LIN {X 0,Y 520.453,Z 702.53,A -85,B 0,C 180,E1 4696.9,E2 4696.9} C_VEL
LIN {X 0,Y 520.349,Z 702.53,A -85,B 0,C 180,E1 4702.128,E2 4702.128} C_VEL
LIN {X 0,Y 520.208,Z 702.53,A -85,B 0,C 180,E1 4707.632,E2 4707.632} C_VEL
LIN {X 0,Y 520.173,Z 702.53,A -85,B 0,C 180,E1 4713.424,E2 4713.424} C_VEL
LIN {X 0,Y 520.246,Z 702.53,A -85,B 0,C 180,E1 4719.624,E2 4719.624} C_VEL
LIN {X 0,Y 520.141,Z 702.53,A -85,B 0,C 180,E1 4725.871,E2 4725.871} C_VEL
LIN {X 0,Y 520.098,Z 702.53,A -85,B 0,C 180,E1 4731.533,E2 4731.533} C_VEL
LIN {X 0,Y 520.321,Z 702.53,A -85,B 0,C 180,E1 4737.206,E2 4737.206} C_VEL
LIN {X 0,Y 520.267,Z 702.53,A -85,B 0,C 180,E1 4742.35,E2 4742.35} C_VEL
LIN {X 0,Y 520.358,Z 702.53,A -85,B 0,C 180,E1 4748.054,E2 4748.054} C_VEL
LIN {X 0,Y 520.437,Z 702.53,A -85,B 0,C 180,E1 4753.145,E2 4753.145} C_VEL
LIN {X 0,Y 520.522,Z 702.53,A -85,B 0,C 180,E1 4758.292,E2 4758.292} C_VEL
LIN {X 0,Y 520.587,Z 702.53,A -85,B 0,C 180,E1 4763.342,E2 4763.342} C_VEL
LIN {X 0,Y 520.67,Z 703.242,A -85,B 0,C 180,E1 4767.374,E2 4767.374} C_VEL
LIN {X 0,Y 530.204,Z 730.276,A -85,B 0,C 180,E1 4768.601,E2 4768.601} C_VEL
LIN {X 0,Y 528.889,Z 767.403,A -85,B 0,C 180,E1 4769.944,E2 4769.944} C_VEL
LIN {X 0,Y 527.056,Z 803.071,A -85,B 0,C 180,E1 4771.949,E2 4771.949} C_VEL
LIN {X 0,Y 525.109,Z 835.334,A -85,B 0,C 180,E1 4774.533,E2 4774.533} C_VEL
LIN {X 0,Y 523.491,Z 864.071,A -85,B 0,C 180,E1 4777.662,E2 4777.662} C_VEL
LIN {X 0,Y 522.246,Z 888.252,A -85,B 0,C 180,E1 4781.228,E2 4781.228} C_VEL
LIN {X 0,Y 521.421,Z 907.192,A -85,B 0,C 180,E1 4785.098,E2 4785.098} C_VEL
LIN {X 0,Y 521.133,Z 919.028,A -85,B 0,C 180,E1 4788.574,E2 4788.574} C_VEL
LIN {X 0,Y 520.904,Z 926.713,A -85,B 0,C 180,E1 4792.124,E2 4792.124} C_VEL
LIN {X 0,Y 520.609,Z 930.33,A -85,B 0,C 180,E1 4796.089,E2 4796.089} C_VEL
LIN {X 0,Y 520.787,Z 928.438,A -85,B 0,C 180,E1 4800.509,E2 4800.509} C_VEL
LIN {X 0,Y 521.135,Z 920.633,A -85,B 0,C 180,E1 4804.748,E2 4804.748} C_VEL
LIN {X 0,Y 521.384,Z 907.878,A -85,B 0,C 180,E1 4808.645,E2 4808.645} C_VEL
LIN {X 0,Y 522.078,Z 890.326,A -85,B 0,C 180,E1 4812.316,E2 4812.316} C_VEL
LIN {X 0,Y 523.248,Z 867.61,A -85,B 0,C 180,E1 4815.79,E2 4815.79} C_VEL
LIN {X 0,Y 524.928,Z 839.521,A -85,B 0,C 180,E1 4818.979,E2 4818.979} C_VEL
LIN {X 0,Y 526.831,Z 807.399,A -85,B 0,C 180,E1 4821.654,E2 4821.654} C_VEL
LIN {X 0,Y 528.689,Z 772.934,A -85,B 0,C 180,E1 4823.704,E2 4823.704} C_VEL
LIN {X 0,Y 530.241,Z 736.63,A -85,B 0,C 180,E1 4825.119,E2 4825.119} C_VEL
LIN {X 0,Y 529.84,Z 727.033,A -85,B 0,C 180,E1 4825.43,E2 4825.43} C_VEL
LIN {X 0,Y 520.271,Z 702.53,A -85,B 0,C 180,E1 4826.686,E2 4826.686} C_VEL
LIN {X 0,Y 520.292,Z 702.53,A -85,B 0,C 180,E1 4832.373,E2 4832.373} C_VEL
LIN {X 0,Y 520.403,Z 702.53,A -85,B 0,C 180,E1 4838.112,E2 4838.112} C_VEL
LIN {X 0,Y 520.549,Z 702.53,A -85,B 0,C 180,E1 4843.167,E2 4843.167} C_VEL
LIN {X 0,Y 520.567,Z 702.53,A -85,B 0,C 180,E1 4848.309,E2 4848.309} C_VEL
LIN {X 0,Y 520.603,Z 702.53,A -85,B 0,C 180,E1 4853.357,E2 4853.357} C_VEL
LIN {X 0,Y 520.62,Z 702.53,A -85,B 0,C 180,E1 4858.353,E2 4858.353} C_VEL
LIN {X 0,Y 520.671,Z 702.53,A -85,B 0,C 180,E1 4863.336,E2 4863.336} C_VEL
LIN {X 0,Y 520.512,Z 702.53,A -85,B 0,C 180,E1 4868.346,E2 4868.346} C_VEL
LIN {X 0,Y 520.449,Z 702.53,A -85,B 0,C 180,E1 4873.423,E2 4873.423} C_VEL
LIN {X 0,Y 520.367,Z 702.53,A -85,B 0,C 180,E1 4878.611,E2 4878.611} C_VEL
LIN {X 0,Y 520.283,Z 702.53,A -85,B 0,C 180,E1 4883.966,E2 4883.966} C_VEL
LIN {X 0,Y 520.16,Z 702.53,A -85,B 0,C 180,E1 4889.558,E2 4889.558} C_VEL
LIN {X 0,Y 520.063,Z 702.53,A -85,B 0,C 180,E1 4894.193,E2 4894.193} C_VEL
LIN {X 0,Y 516.119,Z 702.53,A -85,B 0,C 180,E1 4896.079,E2 4896.079} C_VEL
LIN {X 0,Y 512.277,Z 702.53,A -85,B 0,C 180,E1 4897.994,E2 4897.994} C_VEL
LIN {X 0,Y 512.218,Z 702.53,A -85,B 0,C 180,E1 4902.662,E2 4902.662} C_VEL
LIN {X 0,Y 512.145,Z 702.53,A -85,B 0,C 180,E1 4907.449,E2 4907.449} C_VEL
LIN {X 0,Y 512.253,Z 702.53,A -85,B 0,C 180,E1 4914.109,E2 4914.109} C_VEL
LIN {X 0,Y 527.514,Z 735.275,A -85,B 0,C 180,E1 4915.852,E2 4915.852} C_VEL
LIN {X 0,Y 526.665,Z 780.172,A -85,B 0,C 180,E1 4916.724,E2 4916.724} C_VEL
LIN {X 0,Y 525.012,Z 817.63,A -85,B 0,C 180,E1 4918.058,E2 4918.058} C_VEL
LIN {X 0,Y 522.673,Z 854.221,A -85,B 0,C 180,E1 4920.016,E2 4920.016} C_VEL
LIN {X 0,Y 520.021,Z 889.901,A -85,B 0,C 180,E1 4922.686,E2 4922.686} C_VEL
LIN {X 0,Y 517.692,Z 920.346,A -85,B 0,C 180,E1 4925.724,E2 4925.724} C_VEL
LIN {X 0,Y 515.734,Z 947.246,A -85,B 0,C 180,E1 4929.22,E2 4929.22} C_VEL
LIN {X 0,Y 514.274,Z 970.267,A -85,B 0,C 180,E1 4933.156,E2 4933.156} C_VEL
LIN {X 0,Y 513.457,Z 987.982,A -85,B 0,C 180,E1 4937.266,E2 4937.266} C_VEL
LIN {X 0,Y 513.159,Z 1000.677,A -85,B 0,C 180,E1 4941.545,E2 4941.545} C_VEL
LIN {X 0,Y 512.986,Z 1006.957,A -85,B 0,C 180,E1 4944.937,E2 4944.937} C_VEL
LIN {X 0,Y 513.01,Z 1010.088,A -85,B 0,C 180,E1 4948.314,E2 4948.314} C_VEL
LIN {X 0,Y 513.121,Z 1010.089,A -85,B 0,C 180,E1 4951.685,E2 4951.685} C_VEL
LIN {X 0,Y 513.106,Z 1005.755,A -85,B 0,C 180,E1 4955.908,E2 4955.908} C_VEL
LIN {X 0,Y 513.225,Z 996.305,A -85,B 0,C 180,E1 4960.161,E2 4960.161} C_VEL
LIN {X 0,Y 513.729,Z 982.23,A -85,B 0,C 180,E1 4964.223,E2 4964.223} C_VEL
LIN {X 0,Y 514.773,Z 962.39,A -85,B 0,C 180,E1 4968.322,E2 4968.322} C_VEL
LIN {X 0,Y 516.496,Z 936.317,A -85,B 0,C 180,E1 4972.322,E2 4972.322} C_VEL
LIN {X 0,Y 518.843,Z 905.455,A -85,B 0,C 180,E1 4975.866,E2 4975.866} C_VEL
LIN {X 0,Y 521.362,Z 871.934,A -85,B 0,C 180,E1 4978.763,E2 4978.763} C_VEL
LIN {X 0,Y 523.868,Z 836.553,A -85,B 0,C 180,E1 4981.015,E2 4981.015} C_VEL
LIN {X 0,Y 525.939,Z 799.077,A -85,B 0,C 180,E1 4982.679,E2 4982.679} C_VEL
LIN {X 0,Y 527.422,Z 761.468,A -85,B 0,C 180,E1 4983.701,E2 4983.701} C_VEL
LIN {X 0,Y 526.932,Z 733.943,A -85,B 0,C 180,E1 4984.213,E2 4984.213} C_VEL
LIN {X 0,Y 512.224,Z 702.53,A -85,B 0,C 180,E1 4985.89,E2 4985.89} C_VEL
LIN {X 0,Y 512.283,Z 702.53,A -85,B 0,C 180,E1 4990.395,E2 4990.395} C_VEL
LIN {X 0,Y 512.226,Z 702.53,A -85,B 0,C 180,E1 4995,E2 4995} C_VEL
LIN {X 0,Y 512.163,Z 702.53,A -85,B 0,C 180,E1 5000.001,E2 5000.001} C_VEL
LIN {X 0,Y 512.28,Z 702.53,A -85,B 0,C 180,E1 5005.959,E2 5005.959} C_VEL
LIN {X 0,Y 512.335,Z 702.53,A -85,B 0,C 180,E1 5011.876,E2 5011.876} C_VEL
LIN {X 0,Y 512.348,Z 702.53,A -85,B 0,C 180,E1 5017.478,E2 5017.478} C_VEL
LIN {X 0,Y 512.571,Z 702.53,A -85,B 0,C 180,E1 5022.868,E2 5022.868} C_VEL
LIN {X 0,Y 512.624,Z 702.53,A -85,B 0,C 180,E1 5028.097,E2 5028.097} C_VEL
LIN {X 0,Y 512.715,Z 702.53,A -85,B 0,C 180,E1 5033.227,E2 5033.227} C_VEL
LIN {X 0,Y 512.748,Z 702.53,A -85,B 0,C 180,E1 5038.3,E2 5038.3} C_VEL
LIN {X 0,Y 512.775,Z 702.53,A -85,B 0,C 180,E1 5043.36,E2 5043.36} C_VEL
LIN {X 0,Y 512.629,Z 702.53,A -85,B 0,C 180,E1 5048.448,E2 5048.448} C_VEL
LIN {X 0,Y 512.557,Z 702.53,A -85,B 0,C 180,E1 5053.699,E2 5053.699} C_VEL
LIN {X 0,Y 512.437,Z 702.53,A -85,B 0,C 180,E1 5059.553,E2 5059.553} C_VEL
LIN {X 0,Y 512.378,Z 702.53,A -85,B 0,C 180,E1 5064.33,E2 5064.33} C_VEL
LIN {X 0,Y 512.22,Z 702.53,A -85,B 0,C 180,E1 5070.031,E2 5070.031} C_VEL
LIN {X 0,Y 512.25,Z 702.53,A -85,B 0,C 180,E1 5076.072,E2 5076.072} C_VEL
LIN {X 0,Y 512.334,Z 702.53,A -85,B 0,C 180,E1 5080.361,E2 5080.361} C_VEL
LIN {X 0,Y 512.23,Z 702.53,A -85,B 0,C 180,E1 5085.006,E2 5085.006} C_VEL
LIN {X 0,Y 512.19,Z 702.53,A -85,B 0,C 180,E1 5091.779,E2 5091.779} C_VEL
LIN {X 0,Y 512.381,Z 702.53,A -85,B 0,C 180,E1 5097.987,E2 5097.987} C_VEL
LIN {X 0,Y 512.315,Z 702.53,A -85,B 0,C 180,E1 5103.78,E2 5103.78} C_VEL
LIN {X 0,Y 512.454,Z 702.53,A -85,B 0,C 180,E1 5109.307,E2 5109.307} C_VEL
LIN {X 0,Y 512.576,Z 702.53,A -85,B 0,C 180,E1 5114.636,E2 5114.636} C_VEL
LIN {X 0,Y 512.667,Z 702.53,A -85,B 0,C 180,E1 5119.828,E2 5119.828} C_VEL
LIN {X 0,Y 512.796,Z 702.53,A -85,B 0,C 180,E1 5124.935,E2 5124.935} C_VEL
LIN {X 0,Y 512.85,Z 702.53,A -85,B 0,C 180,E1 5126.814,E2 5126.814} C_VEL
LIN {X 0,Y 523.324,Z 732.22,A -85,B 0,C 180,E1 5128.219,E2 5128.219} C_VEL
LIN {X 0,Y 521.784,Z 768.966,A -85,B 0,C 180,E1 5129.604,E2 5129.604} C_VEL
LIN {X 0,Y 519.712,Z 804.317,A -85,B 0,C 180,E1 5131.664,E2 5131.664} C_VEL
LIN {X 0,Y 517.597,Z 836.301,A -85,B 0,C 180,E1 5134.285,E2 5134.285} C_VEL
LIN {X 0,Y 515.894,Z 863.965,A -85,B 0,C 180,E1 5137.353,E2 5137.353} C_VEL
LIN {X 0,Y 514.506,Z 888.069,A -85,B 0,C 180,E1 5140.952,E2 5140.952} C_VEL
LIN {X 0,Y 513.605,Z 906.585,A -85,B 0,C 180,E1 5144.764,E2 5144.764} C_VEL
LIN {X 0,Y 513.296,Z 918.381,A -85,B 0,C 180,E1 5148.204,E2 5148.204} C_VEL
LIN {X 0,Y 513.083,Z 925.846,A -85,B 0,C 180,E1 5151.513,E2 5151.513} C_VEL
LIN {X 0,Y 512.752,Z 929.432,A -85,B 0,C 180,E1 5154.332,E2 5154.332} C_VEL
LIN {X 0,Y 512.739,Z 930.276,A -85,B 0,C 180,E1 5158.092,E2 5158.092} C_VEL
LIN {X 0,Y 513.008,Z 926.555,A -85,B 0,C 180,E1 5161.97,E2 5161.97} C_VEL
LIN {X 0,Y 513.267,Z 917.534,A -85,B 0,C 180,E1 5166.016,E2 5166.016} C_VEL
LIN {X 0,Y 513.726,Z 902.905,A -85,B 0,C 180,E1 5170.018,E2 5170.018} C_VEL
LIN {X 0,Y 514.711,Z 883.678,A -85,B 0,C 180,E1 5173.698,E2 5173.698} C_VEL
LIN {X 0,Y 516.24,Z 858.437,A -85,B 0,C 180,E1 5177.248,E2 5177.248} C_VEL
LIN {X 0,Y 518.108,Z 829.258,A -85,B 0,C 180,E1 5180.276,E2 5180.276} C_VEL
LIN {X 0,Y 520.21,Z 797.288,A -85,B 0,C 180,E1 5182.71,E2 5182.71} C_VEL
LIN {X 0,Y 522.178,Z 763.148,A -85,B 0,C 180,E1 5184.574,E2 5184.574} C_VEL
LIN {X 0,Y 523.095,Z 729.725,A -85,B 0,C 180,E1 5185.794,E2 5185.794} C_VEL
LIN {X 0,Y 512.376,Z 702.53,A -85,B 0,C 180,E1 5187.187,E2 5187.187} C_VEL
LIN {X 0,Y 512.347,Z 702.53,A -85,B 0,C 180,E1 5193.803,E2 5193.803} C_VEL
LIN {X 0,Y 512.539,Z 702.53,A -85,B 0,C 180,E1 5199.33,E2 5199.33} C_VEL
LIN {X 0,Y 512.692,Z 702.53,A -85,B 0,C 180,E1 5204.657,E2 5204.657} C_VEL
LIN {X 0,Y 512.691,Z 702.53,A -85,B 0,C 180,E1 5209.844,E2 5209.844} C_VEL
LIN {X 0,Y 512.802,Z 702.53,A -85,B 0,C 180,E1 5214.95,E2 5214.95} C_VEL
LIN {X 0,Y 513.033,Z 702.53,A -85,B 0,C 180,E1 5221.699,E2 5221.699} C_VEL
LIN {X 0,Y 512.792,Z 702.53,A -85,B 0,C 180,E1 5226.772,E2 5226.772} C_VEL
LIN {X 0,Y 512.595,Z 702.53,A -85,B 0,C 180,E1 5231.903,E2 5231.903} C_VEL
LIN {X 0,Y 512.513,Z 702.53,A -85,B 0,C 180,E1 5237.134,E2 5237.134} C_VEL
LIN {X 0,Y 512.367,Z 702.53,A -85,B 0,C 180,E1 5242.521,E2 5242.521} C_VEL
LIN {X 0,Y 512.28,Z 702.53,A -85,B 0,C 180,E1 5248.128,E2 5248.128} C_VEL
LIN {X 0,Y 512.158,Z 702.53,A -85,B 0,C 180,E1 5254.412,E2 5254.412} C_VEL
LIN {X 0,Y 512.277,Z 702.53,A -85,B 0,C 180,E1 5257.994,E2 5257.994} C_VEL
LIN {X 0,Y 509.81,Z 702.53,A -85,B 0,C 180,E1 5259.424,E2 5259.424} C_VEL
LIN {X 0,Y 504.22,Z 702.53,A -85,B 0,C 180,E1 5261.814,E2 5261.814} C_VEL
LIN {X 0,Y 504.161,Z 702.53,A -85,B 0,C 180,E1 5268.447,E2 5268.447} C_VEL
LIN {X 0,Y 504.294,Z 703.001,A -85,B 0,C 180,E1 5273.624,E2 5273.624} C_VEL
LIN {X 0,Y 520.902,Z 737.205,A -85,B 0,C 180,E1 5275.388,E2 5275.388} C_VEL
LIN {X 0,Y 519.979,Z 782.48,A -85,B 0,C 180,E1 5276.312,E2 5276.312} C_VEL
LIN {X 0,Y 518.084,Z 819.989,A -85,B 0,C 180,E1 5277.7,E2 5277.7} C_VEL
LIN {X 0,Y 515.587,Z 855.91,A -85,B 0,C 180,E1 5279.682,E2 5279.682} C_VEL
LIN {X 0,Y 512.884,Z 889.628,A -85,B 0,C 180,E1 5282.248,E2 5282.248} C_VEL
LIN {X 0,Y 510.271,Z 920.538,A -85,B 0,C 180,E1 5285.371,E2 5285.371} C_VEL
LIN {X 0,Y 508.143,Z 947.246,A -85,B 0,C 180,E1 5288.895,E2 5288.895} C_VEL
LIN {X 0,Y 506.549,Z 970.266,A -85,B 0,C 180,E1 5292.891,E2 5292.891} C_VEL
LIN {X 0,Y 505.637,Z 987.983,A -85,B 0,C 180,E1 5297.066,E2 5297.066} C_VEL
LIN {X 0,Y 505.266,Z 1000.677,A -85,B 0,C 180,E1 5301.412,E2 5301.412} C_VEL
LIN {X 0,Y 505.093,Z 1006.957,A -85,B 0,C 180,E1 5304.858,E2 5304.858} C_VEL
LIN {X 0,Y 505.108,Z 1010.088,A -85,B 0,C 180,E1 5308.288,E2 5308.288} C_VEL
LIN {X 0,Y 505.214,Z 1010.089,A -85,B 0,C 180,E1 5311.711,E2 5311.711} C_VEL
LIN {X 0,Y 505.215,Z 1005.755,A -85,B 0,C 180,E1 5316.001,E2 5316.001} C_VEL
LIN {X 0,Y 505.339,Z 996.305,A -85,B 0,C 180,E1 5320.321,E2 5320.321} C_VEL
LIN {X 0,Y 505.978,Z 981.123,A -85,B 0,C 180,E1 5324.726,E2 5324.726} C_VEL
LIN {X 0,Y 507.264,Z 959.659,A -85,B 0,C 180,E1 5329.101,E2 5329.101} C_VEL
LIN {X 0,Y 509.1,Z 934.488,A -85,B 0,C 180,E1 5332.91,E2 5332.91} C_VEL
LIN {X 0,Y 511.618,Z 904.312,A -85,B 0,C 180,E1 5336.376,E2 5336.376} C_VEL
LIN {X 0,Y 514.376,Z 870.408,A -85,B 0,C 180,E1 5339.311,E2 5339.311} C_VEL
LIN {X 0,Y 517.13,Z 834.201,A -85,B 0,C 180,E1 5341.6,E2 5341.6} C_VEL
LIN {X 0,Y 519.339,Z 796.328,A -85,B 0,C 180,E1 5343.252,E2 5343.252} C_VEL
LIN {X 0,Y 520.911,Z 757.963,A -85,B 0,C 180,E1 5344.248,E2 5344.248} C_VEL
LIN {X 0,Y 520.337,Z 736.531,A -85,B 0,C 180,E1 5344.666,E2 5344.666} C_VEL
LIN {X 0,Y 504.384,Z 703.582,A -85,B 0,C 180,E1 5346.384,E2 5346.384} C_VEL
LIN {X 0,Y 504.341,Z 702.53,A -85,B 0,C 180,E1 5346.467,E2 5346.467} C_VEL
LIN {X 0,Y 504.271,Z 702.53,A -85,B 0,C 180,E1 5351.567,E2 5351.567} C_VEL
LIN {X 0,Y 504.201,Z 702.53,A -85,B 0,C 180,E1 5356.493,E2 5356.493} C_VEL
LIN {X 0,Y 504.233,Z 702.53,A -85,B 0,C 180,E1 5363.227,E2 5363.227} C_VEL
LIN {X 0,Y 504.452,Z 702.53,A -85,B 0,C 180,E1 5369.425,E2 5369.425} C_VEL
LIN {X 0,Y 504.393,Z 702.53,A -85,B 0,C 180,E1 5375.229,E2 5375.229} C_VEL
LIN {X 0,Y 504.575,Z 702.53,A -85,B 0,C 180,E1 5380.784,E2 5380.784} C_VEL
LIN {X 0,Y 504.766,Z 702.53,A -85,B 0,C 180,E1 5386.152,E2 5386.152} C_VEL
LIN {X 0,Y 504.81,Z 702.53,A -85,B 0,C 180,E1 5391.392,E2 5391.392} C_VEL
LIN {X 0,Y 505.024,Z 702.53,A -85,B 0,C 180,E1 5396.561,E2 5396.561} C_VEL
LIN {X 0,Y 505.115,Z 702.53,A -85,B 0,C 180,E1 5401.698,E2 5401.698} C_VEL
LIN {X 0,Y 504.886,Z 702.53,A -85,B 0,C 180,E1 5406.851,E2 5406.851} C_VEL
LIN {X 0,Y 504.703,Z 702.53,A -85,B 0,C 180,E1 5412.064,E2 5412.064} C_VEL
LIN {X 0,Y 504.627,Z 702.53,A -85,B 0,C 180,E1 5417.381,E2 5417.381} C_VEL
LIN {X 0,Y 504.481,Z 702.53,A -85,B 0,C 180,E1 5422.863,E2 5422.863} C_VEL
LIN {X 0,Y 504.304,Z 702.53,A -85,B 0,C 180,E1 5428.582,E2 5428.582} C_VEL
LIN {X 0,Y 504.294,Z 702.53,A -85,B 0,C 180,E1 5434.623,E2 5434.623} C_VEL
LIN {X 0,Y 504.327,Z 702.53,A -85,B 0,C 180,E1 5441.138,E2 5441.138} C_VEL
LIN {X 0,Y 504.182,Z 702.53,A -85,B 0,C 180,E1 5446.497,E2 5446.497} C_VEL
LIN {X 0,Y 504.301,Z 702.53,A -85,B 0,C 180,E1 5453.24,E2 5453.24} C_VEL
LIN {X 0,Y 504.456,Z 702.53,A -85,B 0,C 180,E1 5459.434,E2 5459.434} C_VEL
LIN {X 0,Y 504.423,Z 702.53,A -85,B 0,C 180,E1 5465.24,E2 5465.24} C_VEL
LIN {X 0,Y 504.568,Z 702.53,A -85,B 0,C 180,E1 5470.793,E2 5470.793} C_VEL
LIN {X 0,Y 504.732,Z 702.53,A -85,B 0,C 180,E1 5476.162,E2 5476.162} C_VEL
LIN {X 0,Y 504.81,Z 702.53,A -85,B 0,C 180,E1 5481.404,E2 5481.404} C_VEL
LIN {X 0,Y 504.939,Z 702.53,A -85,B 0,C 180,E1 5486.252,E2 5486.252} C_VEL
LIN {X 0,Y 516.47,Z 735.654,A -85,B 0,C 180,E1 5487.871,E2 5487.871} C_VEL
LIN {X 0,Y 514.64,Z 773.223,A -85,B 0,C 180,E1 5489.37,E2 5489.37} C_VEL
LIN {X 0,Y 512.364,Z 806.818,A -85,B 0,C 180,E1 5491.434,E2 5491.434} C_VEL
LIN {X 0,Y 509.935,Z 840.525,A -85,B 0,C 180,E1 5494.349,E2 5494.349} C_VEL
LIN {X 0,Y 507.942,Z 868.69,A -85,B 0,C 180,E1 5497.683,E2 5497.683} C_VEL
LIN {X 0,Y 506.529,Z 891.604,A -85,B 0,C 180,E1 5501.346,E2 5501.346} C_VEL
LIN {X 0,Y 505.704,Z 908.552,A -85,B 0,C 180,E1 5505.067,E2 5505.067} C_VEL
LIN {X 0,Y 505.306,Z 921.279,A -85,B 0,C 180,E1 5509.178,E2 5509.178} C_VEL
LIN {X 0,Y 504.987,Z 927.955,A -85,B 0,C 180,E1 5512.86,E2 5512.86} C_VEL
LIN {X 0,Y 504.77,Z 930.444,A -85,B 0,C 180,E1 5516.643,E2 5516.643} C_VEL
LIN {X 0,Y 504.964,Z 928.525,A -85,B 0,C 180,E1 5520.533,E2 5520.533} C_VEL
LIN {X 0,Y 505.339,Z 921.644,A -85,B 0,C 180,E1 5524.567,E2 5524.567} C_VEL
LIN {X 0,Y 505.69,Z 908.702,A -85,B 0,C 180,E1 5528.804,E2 5528.804} C_VEL
LIN {X 0,Y 506.492,Z 891.874,A -85,B 0,C 180,E1 5532.515,E2 5532.515} C_VEL
LIN {X 0,Y 507.843,Z 869.857,A -85,B 0,C 180,E1 5536.066,E2 5536.066} C_VEL
LIN {X 0,Y 509.836,Z 842.048,A -85,B 0,C 180,E1 5539.4,E2 5539.4} C_VEL
LIN {X 0,Y 512.24,Z 809.508,A -85,B 0,C 180,E1 5542.28,E2 5542.28} C_VEL
LIN {X 0,Y 514.549,Z 776.365,A -85,B 0,C 180,E1 5544.383,E2 5544.383} C_VEL
LIN {X 0,Y 516.429,Z 741.237,A -85,B 0,C 180,E1 5545.873,E2 5545.873} C_VEL
LIN {X 0,Y 516.124,Z 731.683,A -85,B 0,C 180,E1 5546.208,E2 5546.208} C_VEL
LIN {X 0,Y 504.467,Z 702.53,A -85,B 0,C 180,E1 5547.785,E2 5547.785} C_VEL
LIN {X 0,Y 504.444,Z 702.53,A -85,B 0,C 180,E1 5553.824,E2 5553.824} C_VEL
LIN {X 0,Y 504.577,Z 702.53,A -85,B 0,C 180,E1 5558.989,E2 5558.989} C_VEL
LIN {X 0,Y 504.754,Z 702.53,A -85,B 0,C 180,E1 5564.409,E2 5564.409} C_VEL
LIN {X 0,Y 504.749,Z 702.53,A -85,B 0,C 180,E1 5570.607,E2 5570.607} C_VEL
LIN {X 0,Y 504.959,Z 702.53,A -85,B 0,C 180,E1 5576.588,E2 5576.588} C_VEL
LIN {X 0,Y 505.122,Z 702.53,A -85,B 0,C 180,E1 5581.725,E2 5581.725} C_VEL
LIN {X 0,Y 504.866,Z 702.53,A -85,B 0,C 180,E1 5586.879,E2 5586.879} C_VEL
LIN {X 0,Y 504.675,Z 702.53,A -85,B 0,C 180,E1 5592.093,E2 5592.093} C_VEL
LIN {X 0,Y 504.584,Z 702.53,A -85,B 0,C 180,E1 5597.411,E2 5597.411} C_VEL
LIN {X 0,Y 504.438,Z 702.53,A -85,B 0,C 180,E1 5602.895,E2 5602.895} C_VEL
LIN {X 0,Y 504.305,Z 702.53,A -85,B 0,C 180,E1 5608.613,E2 5608.613} C_VEL
LIN {X 0,Y 504.259,Z 702.53,A -85,B 0,C 180,E1 5614.659,E2 5614.659} C_VEL
LIN {X 0,Y 504.37,Z 702.53,A -85,B 0,C 180,E1 5618.931,E2 5618.931} C_VEL
LIN {X 0,Y 504.22,Z 702.53,A -85,B 0,C 180,E1 5621.814,E2 5621.814} C_VEL
LIN {X 0,Y 500.216,Z 702.53,A -85,B 0,C 180,E1 5623.761,E2 5623.761} C_VEL
LIN {X 0,Y 496.244,Z 702.53,A -85,B 0,C 180,E1 5625.739,E2 5625.739} C_VEL
LIN {X 0,Y 496.248,Z 702.53,A -85,B 0,C 180,E1 5632.249,E2 5632.249} C_VEL
LIN {X 0,Y 496.355,Z 703.123,A -85,B 0,C 180,E1 5633.023,E2 5633.023} C_VEL
LIN {X 0,Y 514.359,Z 740.401,A -85,B 0,C 180,E1 5634.96,E2 5634.96} C_VEL
LIN {X 0,Y 513.356,Z 783.291,A -85,B 0,C 180,E1 5635.845,E2 5635.845} C_VEL
LIN {X 0,Y 511.356,Z 819.987,A -85,B 0,C 180,E1 5637.222,E2 5637.222} C_VEL
LIN {X 0,Y 508.736,Z 855.33,A -85,B 0,C 180,E1 5639.187,E2 5639.187} C_VEL
LIN {X 0,Y 505.64,Z 890.368,A -85,B 0,C 180,E1 5641.887,E2 5641.887} C_VEL
LIN {X 0,Y 502.751,Z 921.941,A -85,B 0,C 180,E1 5645.152,E2 5645.152} C_VEL
LIN {X 0,Y 500.446,Z 948.698,A -85,B 0,C 180,E1 5648.786,E2 5648.786} C_VEL
LIN {X 0,Y 498.724,Z 971.345,A -85,B 0,C 180,E1 5652.841,E2 5652.841} C_VEL
LIN {X 0,Y 497.807,Z 987.983,A -85,B 0,C 180,E1 5656.859,E2 5656.859} C_VEL
LIN {X 0,Y 497.391,Z 1000.677,A -85,B 0,C 180,E1 5661.275,E2 5661.275} C_VEL
LIN {X 0,Y 497.201,Z 1006.957,A -85,B 0,C 180,E1 5664.776,E2 5664.776} C_VEL
LIN {X 0,Y 497.232,Z 1010.088,A -85,B 0,C 180,E1 5668.261,E2 5668.261} C_VEL
LIN {X 0,Y 497.311,Z 1010.089,A -85,B 0,C 180,E1 5671.739,E2 5671.739} C_VEL
LIN {X 0,Y 497.337,Z 1005.755,A -85,B 0,C 180,E1 5676.096,E2 5676.096} C_VEL
LIN {X 0,Y 497.452,Z 996.305,A -85,B 0,C 180,E1 5680.487,E2 5680.487} C_VEL
LIN {X 0,Y 498.221,Z 980.677,A -85,B 0,C 180,E1 5685.076,E2 5685.076} C_VEL
LIN {X 0,Y 499.611,Z 959.657,A -85,B 0,C 180,E1 5689.405,E2 5689.405} C_VEL
LIN {X 0,Y 501.625,Z 934.487,A -85,B 0,C 180,E1 5693.271,E2 5693.271} C_VEL
LIN {X 0,Y 504.349,Z 904.421,A -85,B 0,C 180,E1 5696.775,E2 5696.775} C_VEL
LIN {X 0,Y 507.362,Z 870.397,A -85,B 0,C 180,E1 5699.757,E2 5699.757} C_VEL
LIN {X 0,Y 510.264,Z 835.023,A -85,B 0,C 180,E1 5702.027,E2 5702.027} C_VEL
LIN {X 0,Y 512.682,Z 796.685,A -85,B 0,C 180,E1 5703.727,E2 5703.727} C_VEL
LIN {X 0,Y 514.323,Z 759.781,A -85,B 0,C 180,E1 5704.704,E2 5704.704} C_VEL
LIN {X 0,Y 514.024,Z 739.721,A -85,B 0,C 180,E1 5705.078,E2 5705.078} C_VEL
LIN {X 0,Y 496.538,Z 704.023,A -85,B 0,C 180,E1 5706.985,E2 5706.985} C_VEL
LIN {X 0,Y 496.377,Z 702.53,A -85,B 0,C 180,E1 5707.084,E2 5707.084} C_VEL
LIN {X 0,Y 496.33,Z 702.53,A -85,B 0,C 180,E1 5713.134,E2 5713.134} C_VEL
LIN {X 0,Y 496.224,Z 702.53,A -85,B 0,C 180,E1 5719.486,E2 5719.486} C_VEL
LIN {X 0,Y 496.41,Z 702.53,A -85,B 0,C 180,E1 5725.161,E2 5725.161} C_VEL
LIN {X 0,Y 496.498,Z 702.53,A -85,B 0,C 180,E1 5730.894,E2 5730.894} C_VEL
LIN {X 0,Y 496.474,Z 702.53,A -85,B 0,C 180,E1 5736.716,E2 5736.716} C_VEL
LIN {X 0,Y 496.711,Z 702.53,A -85,B 0,C 180,E1 5742.304,E2 5742.304} C_VEL
LIN {X 0,Y 496.798,Z 702.53,A -85,B 0,C 180,E1 5747.712,E2 5747.712} C_VEL
LIN {X 0,Y 496.919,Z 702.53,A -85,B 0,C 180,E1 5753.011,E2 5753.011} C_VEL
LIN {X 0,Y 496.971,Z 702.53,A -85,B 0,C 180,E1 5758.246,E2 5758.246} C_VEL
LIN {X 0,Y 496.985,Z 702.53,A -85,B 0,C 180,E1 5763.467,E2 5763.467} C_VEL
LIN {X 0,Y 496.824,Z 702.53,A -85,B 0,C 180,E1 5768.719,E2 5768.719} C_VEL
LIN {X 0,Y 496.753,Z 702.53,A -85,B 0,C 180,E1 5774.047,E2 5774.047} C_VEL
LIN {X 0,Y 496.608,Z 702.53,A -85,B 0,C 180,E1 5779.613,E2 5779.613} C_VEL
LIN {X 0,Y 496.491,Z 702.53,A -85,B 0,C 180,E1 5785.161,E2 5785.161} C_VEL
LIN {X 0,Y 496.305,Z 702.53,A -85,B 0,C 180,E1 5791.642,E2 5791.642} C_VEL
LIN {X 0,Y 496.394,Z 702.53,A -85,B 0,C 180,E1 5797.778,E2 5797.778} C_VEL
LIN {X 0,Y 496.35,Z 702.53,A -85,B 0,C 180,E1 5804.335,E2 5804.335} C_VEL
LIN {X 0,Y 496.268,Z 702.53,A -85,B 0,C 180,E1 5810.316,E2 5810.316} C_VEL
LIN {X 0,Y 496.451,Z 702.53,A -85,B 0,C 180,E1 5816.83,E2 5816.83} C_VEL
LIN {X 0,Y 496.443,Z 702.53,A -85,B 0,C 180,E1 5822.874,E2 5822.874} C_VEL
LIN {X 0,Y 496.588,Z 702.53,A -85,B 0,C 180,E1 5828.614,E2 5828.614} C_VEL
LIN {X 0,Y 496.74,Z 702.53,A -85,B 0,C 180,E1 5834.133,E2 5834.133} C_VEL
LIN {X 0,Y 496.82,Z 702.53,A -85,B 0,C 180,E1 5839.5,E2 5839.5} C_VEL
LIN {X 0,Y 497.014,Z 702.53,A -85,B 0,C 180,E1 5845.668,E2 5845.668} C_VEL
LIN {X 0,Y 509.668,Z 736.834,A -85,B 0,C 180,E1 5847.445,E2 5847.445} C_VEL
LIN {X 0,Y 507.739,Z 773.59,A -85,B 0,C 180,E1 5848.936,E2 5848.936} C_VEL
LIN {X 0,Y 505.268,Z 807.581,A -85,B 0,C 180,E1 5851.051,E2 5851.051} C_VEL
LIN {X 0,Y 502.691,Z 838.613,A -85,B 0,C 180,E1 5853.765,E2 5853.765} C_VEL
LIN {X 0,Y 500.326,Z 868.599,A -85,B 0,C 180,E1 5857.365,E2 5857.365} C_VEL
LIN {X 0,Y 498.862,Z 890.969,A -85,B 0,C 180,E1 5860.981,E2 5860.981} C_VEL
LIN {X 0,Y 497.859,Z 908.951,A -85,B 0,C 180,E1 5864.979,E2 5864.979} C_VEL
LIN {X 0,Y 497.423,Z 921.235,A -85,B 0,C 180,E1 5869.034,E2 5869.034} C_VEL
LIN {X 0,Y 497.004,Z 928.456,A -85,B 0,C 180,E1 5873.248,E2 5873.248} C_VEL
LIN {X 0,Y 496.83,Z 930.476,A -85,B 0,C 180,E1 5877.104,E2 5877.104} C_VEL
LIN {X 0,Y 497.132,Z 928.024,A -85,B 0,C 180,E1 5881.066,E2 5881.066} C_VEL
LIN {X 0,Y 497.463,Z 920.443,A -85,B 0,C 180,E1 5885.195,E2 5885.195} C_VEL
LIN {X 0,Y 497.847,Z 908.165,A -85,B 0,C 180,E1 5889.131,E2 5889.131} C_VEL
LIN {X 0,Y 498.813,Z 890.154,A -85,B 0,C 180,E1 5893.083,E2 5893.083} C_VEL
LIN {X 0,Y 500.394,Z 867.282,A -85,B 0,C 180,E1 5896.732,E2 5896.732} C_VEL
LIN {X 0,Y 502.837,Z 837.862,A -85,B 0,C 180,E1 5900.225,E2 5900.225} C_VEL
LIN {X 0,Y 505.373,Z 807.979,A -85,B 0,C 180,E1 5902.842,E2 5902.842} C_VEL
LIN {X 0,Y 507.766,Z 775.341,A -85,B 0,C 180,E1 5904.9,E2 5904.9} C_VEL
LIN {X 0,Y 509.831,Z 739.442,A -85,B 0,C 180,E1 5906.399,E2 5906.399} C_VEL
LIN {X 0,Y 508.542,Z 731.945,A -85,B 0,C 180,E1 5906.732,E2 5906.732} C_VEL
LIN {X 0,Y 496.527,Z 702.53,A -85,B 0,C 180,E1 5908.317,E2 5908.317} C_VEL
LIN {X 0,Y 496.521,Z 702.53,A -85,B 0,C 180,E1 5914.84,E2 5914.84} C_VEL
LIN {X 0,Y 496.697,Z 702.53,A -85,B 0,C 180,E1 5920.496,E2 5920.496} C_VEL
LIN {X 0,Y 496.941,Z 702.53,A -85,B 0,C 180,E1 5926.343,E2 5926.343} C_VEL
LIN {X 0,Y 496.897,Z 702.53,A -85,B 0,C 180,E1 5933.038,E2 5933.038} C_VEL
LIN {X 0,Y 496.947,Z 702.53,A -85,B 0,C 180,E1 5938.274,E2 5938.274} C_VEL
LIN {X 0,Y 496.987,Z 702.53,A -85,B 0,C 180,E1 5943.495,E2 5943.495} C_VEL
LIN {X 0,Y 496.802,Z 702.53,A -85,B 0,C 180,E1 5948.748,E2 5948.748} C_VEL
LIN {X 0,Y 496.684,Z 702.53,A -85,B 0,C 180,E1 5954.078,E2 5954.078} C_VEL
LIN {X 0,Y 496.589,Z 702.53,A -85,B 0,C 180,E1 5959.605,E2 5959.605} C_VEL
LIN {X 0,Y 496.496,Z 702.53,A -85,B 0,C 180,E1 5965.192,E2 5965.192} C_VEL
LIN {X 0,Y 496.288,Z 702.53,A -85,B 0,C 180,E1 5971.638,E2 5971.638} C_VEL
LIN {X 0,Y 496.354,Z 702.53,A -85,B 0,C 180,E1 5977.771,E2 5977.771} C_VEL
LIN {X 0,Y 496.295,Z 702.53,A -85,B 0,C 180,E1 5983.135,E2 5983.135} C_VEL
LIN {X 0,Y 496.244,Z 702.53,A -85,B 0,C 180,E1 5985.739,E2 5985.739} C_VEL
LIN {X 0,Y 492.28,Z 702.53,A -85,B 0,C 180,E1 5987.714,E2 5987.714} C_VEL
LIN {X 0,Y 488.305,Z 702.53,A -85,B 0,C 180,E1 5989.72,E2 5989.72} C_VEL
LIN {X 0,Y 488.359,Z 702.618,A -85,B 0,C 180,E1 5992.384,E2 5992.384} C_VEL
LIN {X 0,Y 503.509,Z 734.112,A -85,B 0,C 180,E1 5994.082,E2 5994.082} C_VEL
LIN {X 0,Y 507.653,Z 744.179,A -85,B 0,C 180,E1 5994.548,E2 5994.548} C_VEL
LIN {X 0,Y 506.39,Z 787.879,A -85,B 0,C 180,E1 5995.514,E2 5995.514} C_VEL
LIN {X 0,Y 504.067,Z 828.627,A -85,B 0,C 180,E1 5997.155,E2 5997.155} C_VEL
LIN {X 0,Y 500.888,Z 865.801,A -85,B 0,C 180,E1 5999.443,E2 5999.443} C_VEL
LIN {X 0,Y 497.585,Z 899.748,A -85,B 0,C 180,E1 6002.333,E2 6002.333} C_VEL
LIN {X 0,Y 494.723,Z 929.107,A -85,B 0,C 180,E1 6005.648,E2 6005.648} C_VEL
LIN {X 0,Y 492.305,Z 954.586,A -85,B 0,C 180,E1 6009.398,E2 6009.398} C_VEL
LIN {X 0,Y 490.615,Z 975.708,A -85,B 0,C 180,E1 6013.509,E2 6013.509} C_VEL
LIN {X 0,Y 489.744,Z 992.4,A -85,B 0,C 180,E1 6017.995,E2 6017.995} C_VEL
LIN {X 0,Y 489.461,Z 1002.594,A -85,B 0,C 180,E1 6022.025,E2 6022.025} C_VEL
LIN {X 0,Y 489.332,Z 1008.908,A -85,B 0,C 180,E1 6026.464,E2 6026.464} C_VEL
LIN {X 0,Y 489.328,Z 1010.5,A -85,B 0,C 180,E1 6030,E2 6030} C_VEL
LIN {X 0,Y 489.292,Z 1008.911,A -85,B 0,C 180,E1 6033.536,E2 6033.536} C_VEL
LIN {X 0,Y 489.478,Z 1002.597,A -85,B 0,C 180,E1 6037.974,E2 6037.974} C_VEL
LIN {X 0,Y 489.911,Z 991.043,A -85,B 0,C 180,E1 6042.451,E2 6042.451} C_VEL
LIN {X 0,Y 490.903,Z 973.905,A -85,B 0,C 180,E1 6046.895,E2 6046.895} C_VEL
LIN {X 0,Y 492.715,Z 950.754,A -85,B 0,C 180,E1 6051.23,E2 6051.23} C_VEL
LIN {X 0,Y 495.193,Z 923.794,A -85,B 0,C 180,E1 6055.02,E2 6055.02} C_VEL
LIN {X 0,Y 498.192,Z 893.329,A -85,B 0,C 180,E1 6058.281,E2 6058.281} C_VEL
LIN {X 0,Y 501.466,Z 858.738,A -85,B 0,C 180,E1 6061.056,E2 6061.056} C_VEL
LIN {X 0,Y 504.295,Z 823.807,A -85,B 0,C 180,E1 6063.081,E2 6063.081} C_VEL
LIN {X 0,Y 506.572,Z 783.98,A -85,B 0,C 180,E1 6064.605,E2 6064.605} C_VEL
LIN {X 0,Y 507.422,Z 742.338,A -85,B 0,C 180,E1 6065.512,E2 6065.512} C_VEL
LIN {X 0,Y 488.462,Z 702.53,A -85,B 0,C 180,E1 6067.757,E2 6067.757} C_VEL
LIN {X 0,Y 488.417,Z 702.53,A -85,B 0,C 180,E1 6072.821,E2 6072.821} C_VEL
LIN {X 0,Y 488.356,Z 702.53,A -85,B 0,C 180,E1 6077.868,E2 6077.868} C_VEL
LIN {X 0,Y 488.362,Z 702.53,A -85,B 0,C 180,E1 6084.041,E2 6084.041} C_VEL
LIN {X 0,Y 488.51,Z 702.53,A -85,B 0,C 180,E1 6089.874,E2 6089.874} C_VEL
LIN {X 0,Y 488.558,Z 702.53,A -85,B 0,C 180,E1 6096.316,E2 6096.316} C_VEL
LIN {X 0,Y 488.763,Z 702.53,A -85,B 0,C 180,E1 6102.006,E2 6102.006} C_VEL
LIN {X 0,Y 488.903,Z 702.53,A -85,B 0,C 180,E1 6107.511,E2 6107.511} C_VEL
LIN {X 0,Y 489.004,Z 702.53,A -85,B 0,C 180,E1 6112.897,E2 6112.897} C_VEL
LIN {X 0,Y 489.071,Z 702.53,A -85,B 0,C 180,E1 6118.218,E2 6118.218} C_VEL
LIN {X 0,Y 489.079,Z 702.53,A -85,B 0,C 180,E1 6123.523,E2 6123.523} C_VEL
LIN {X 0,Y 488.896,Z 702.53,A -85,B 0,C 180,E1 6128.993,E2 6128.993} C_VEL
LIN {X 0,Y 488.819,Z 702.53,A -85,B 0,C 180,E1 6134.28,E2 6134.28} C_VEL
LIN {X 0,Y 488.7,Z 702.53,A -85,B 0,C 180,E1 6139.836,E2 6139.836} C_VEL
LIN {X 0,Y 488.52,Z 702.53,A -85,B 0,C 180,E1 6145.601,E2 6145.601} C_VEL
LIN {X 0,Y 488.404,Z 702.53,A -85,B 0,C 180,E1 6151.66,E2 6151.66} C_VEL
LIN {X 0,Y 488.471,Z 702.53,A -85,B 0,C 180,E1 6158.131,E2 6158.131} C_VEL
LIN {X 0,Y 488.441,Z 702.53,A -85,B 0,C 180,E1 6164.718,E2 6164.718} C_VEL
LIN {X 0,Y 488.346,Z 702.53,A -85,B 0,C 180,E1 6170.542,E2 6170.542} C_VEL
LIN {X 0,Y 488.538,Z 702.53,A -85,B 0,C 180,E1 6176.465,E2 6176.465} C_VEL
LIN {X 0,Y 488.527,Z 702.53,A -85,B 0,C 180,E1 6182.397,E2 6182.397} C_VEL
LIN {X 0,Y 488.636,Z 702.53,A -85,B 0,C 180,E1 6188.248,E2 6188.248} C_VEL
LIN {X 0,Y 488.796,Z 702.53,A -85,B 0,C 180,E1 6193.868,E2 6193.868} C_VEL
LIN {X 0,Y 488.908,Z 702.53,A -85,B 0,C 180,E1 6199.328,E2 6199.328} C_VEL
LIN {X 0,Y 489.11,Z 702.994,A -85,B 0,C 180,E1 6205.089,E2 6205.089} C_VEL
LIN {X 0,Y 502.858,Z 738.427,A -85,B 0,C 180,E1 6207.019,E2 6207.019} C_VEL
LIN {X 0,Y 500.702,Z 775.979,A -85,B 0,C 180,E1 6208.597,E2 6208.597} C_VEL
LIN {X 0,Y 498.041,Z 810.216,A -85,B 0,C 180,E1 6210.799,E2 6210.799} C_VEL
LIN {X 0,Y 495.159,Z 842.262,A -85,B 0,C 180,E1 6213.713,E2 6213.713} C_VEL
LIN {X 0,Y 492.788,Z 868.802,A -85,B 0,C 180,E1 6217.036,E2 6217.036} C_VEL
LIN {X 0,Y 490.869,Z 893.86,A -85,B 0,C 180,E1 6221.279,E2 6221.279} C_VEL
LIN {X 0,Y 489.931,Z 910.33,A -85,B 0,C 180,E1 6225.178,E2 6225.178} C_VEL
LIN {X 0,Y 489.529,Z 922.198,A -85,B 0,C 180,E1 6229.353,E2 6229.353} C_VEL
LIN {X 0,Y 489.046,Z 928.902,A -85,B 0,C 180,E1 6233.649,E2 6233.649} C_VEL
LIN {X 0,Y 488.933,Z 930.385,A -85,B 0,C 180,E1 6237.578,E2 6237.578} C_VEL
LIN {X 0,Y 489.26,Z 927.359,A -85,B 0,C 180,E1 6241.624,E2 6241.624} C_VEL
LIN {X 0,Y 489.612,Z 919.117,A -85,B 0,C 180,E1 6245.845,E2 6245.845} C_VEL
LIN {X 0,Y 490.136,Z 905.765,A -85,B 0,C 180,E1 6249.953,E2 6249.953} C_VEL
LIN {X 0,Y 491.382,Z 886.412,A -85,B 0,C 180,E1 6254.041,E2 6254.041} C_VEL
LIN {X 0,Y 493.45,Z 861.845,A -85,B 0,C 180,E1 6257.854,E2 6257.854} C_VEL
LIN {X 0,Y 496.089,Z 833.142,A -85,B 0,C 180,E1 6261.154,E2 6261.154} C_VEL
LIN {X 0,Y 499.011,Z 800.604,A -85,B 0,C 180,E1 6263.839,E2 6263.839} C_VEL
LIN {X 0,Y 501.454,Z 767.586,A -85,B 0,C 180,E1 6265.761,E2 6265.761} C_VEL
LIN {X 0,Y 502.482,Z 736.26,A -85,B 0,C 180,E1 6267.031,E2 6267.031} C_VEL
LIN {X 0,Y 488.596,Z 702.53,A -85,B 0,C 180,E1 6268.957,E2 6268.957} C_VEL
LIN {X 0,Y 488.557,Z 702.53,A -85,B 0,C 180,E1 6274.401,E2 6274.401} C_VEL
LIN {X 0,Y 488.774,Z 702.53,A -85,B 0,C 180,E1 6280.167,E2 6280.167} C_VEL
LIN {X 0,Y 488.988,Z 702.53,A -85,B 0,C 180,E1 6285.725,E2 6285.725} C_VEL
LIN {X 0,Y 488.98,Z 702.53,A -85,B 0,C 180,E1 6291.14,E2 6291.14} C_VEL
LIN {X 0,Y 489.148,Z 702.53,A -85,B 0,C 180,E1 6296.478,E2 6296.478} C_VEL
LIN {X 0,Y 489.327,Z 702.53,A -85,B 0,C 180,E1 6301.781,E2 6301.781} C_VEL
LIN {X 0,Y 489.039,Z 702.53,A -85,B 0,C 180,E1 6307.103,E2 6307.103} C_VEL
LIN {X 0,Y 488.841,Z 702.53,A -85,B 0,C 180,E1 6312.491,E2 6312.491} C_VEL
LIN {X 0,Y 488.696,Z 702.53,A -85,B 0,C 180,E1 6317.997,E2 6317.997} C_VEL
LIN {X 0,Y 488.567,Z 702.53,A -85,B 0,C 180,E1 6323.683,E2 6323.683} C_VEL
LIN {X 0,Y 488.368,Z 702.53,A -85,B 0,C 180,E1 6330.096,E2 6330.096} C_VEL
LIN {X 0,Y 488.406,Z 702.53,A -85,B 0,C 180,E1 6336.551,E2 6336.551} C_VEL
LIN {X 0,Y 488.39,Z 702.53,A -85,B 0,C 180,E1 6342.831,E2 6342.831} C_VEL
LIN {X 0,Y 488.323,Z 702.53,A -85,B 0,C 180,E1 6349.537,E2 6349.537} C_VEL
LIN {X 0,Y 488.305,Z 702.53,A -85,B 0,C 180,E1 6349.72,E2 6349.72} C_VEL
LIN {X 0,Y 484.432,Z 702.53,A -85,B 0,C 180,E1 6350.677,E2 6350.677} C_VEL
LIN {X 0,Y 480.428,Z 702.53,A -85,B 0,C 180,E1 6351.649,E2 6351.649} C_VEL
LIN {X 0,Y 500.884,Z 744.93,A -85,B 0,C 180,E1 6354.069,E2 6354.069} C_VEL
LIN {X 0,Y 499.587,Z 788.838,A -85,B 0,C 180,E1 6355.076,E2 6355.076} C_VEL
LIN {X 0,Y 497.054,Z 829.35,A -85,B 0,C 180,E1 6356.753,E2 6356.753} C_VEL
LIN {X 0,Y 493.909,Z 865.965,A -85,B 0,C 180,E1 6358.985,E2 6358.985} C_VEL
LIN {X 0,Y 490.533,Z 898.836,A -85,B 0,C 180,E1 6361.802,E2 6361.802} C_VEL
LIN {X 0,Y 487.292,Z 929.361,A -85,B 0,C 180,E1 6365.287,E2 6365.287} C_VEL
LIN {X 0,Y 484.603,Z 955.526,A -85,B 0,C 180,E1 6369.226,E2 6369.226} C_VEL
LIN {X 0,Y 482.857,Z 975.874,A -85,B 0,C 180,E1 6373.275,E2 6373.275} C_VEL
LIN {X 0,Y 481.91,Z 992.4,A -85,B 0,C 180,E1 6377.797,E2 6377.797} C_VEL
LIN {X 0,Y 481.567,Z 1002.594,A -85,B 0,C 180,E1 6381.893,E2 6381.893} C_VEL
LIN {X 0,Y 481.43,Z 1008.908,A -85,B 0,C 180,E1 6386.406,E2 6386.406} C_VEL
LIN {X 0,Y 481.439,Z 1010.5,A -85,B 0,C 180,E1 6390,E2 6390} C_VEL
LIN {X 0,Y 481.399,Z 1008.911,A -85,B 0,C 180,E1 6393.594,E2 6393.594} C_VEL
LIN {X 0,Y 481.589,Z 1002.597,A -85,B 0,C 180,E1 6398.106,E2 6398.106} C_VEL
LIN {X 0,Y 482.143,Z 989.856,A -85,B 0,C 180,E1 6403.012,E2 6403.012} C_VEL
LIN {X 0,Y 483.251,Z 972.455,A -85,B 0,C 180,E1 6407.485,E2 6407.485} C_VEL
LIN {X 0,Y 485.158,Z 950.442,A -85,B 0,C 180,E1 6411.628,E2 6411.628} C_VEL
LIN {X 0,Y 487.811,Z 923.856,A -85,B 0,C 180,E1 6415.418,E2 6415.418} C_VEL
LIN {X 0,Y 491.078,Z 893.601,A -85,B 0,C 180,E1 6418.701,E2 6418.701} C_VEL
LIN {X 0,Y 494.353,Z 860.669,A -85,B 0,C 180,E1 6421.388,E2 6421.388} C_VEL
LIN {X 0,Y 497.48,Z 822.598,A -85,B 0,C 180,E1 6423.594,E2 6423.594} C_VEL
LIN {X 0,Y 499.882,Z 783.418,A -85,B 0,C 180,E1 6425.099,E2 6425.099} C_VEL
LIN {X 0,Y 500.617,Z 744.618,A -85,B 0,C 180,E1 6425.981,E2 6425.981} C_VEL
LIN {X 0,Y 480.531,Z 702.53,A -85,B 0,C 180,E1 6428.378,E2 6428.378} C_VEL
LIN {X 0,Y 480.489,Z 702.53,A -85,B 0,C 180,E1 6433.745,E2 6433.745} C_VEL
LIN {X 0,Y 480.423,Z 702.53,A -85,B 0,C 180,E1 6438.925,E2 6438.925} C_VEL
LIN {X 0,Y 480.489,Z 702.53,A -85,B 0,C 180,E1 6445.568,E2 6445.568} C_VEL
LIN {X 0,Y 480.57,Z 702.53,A -85,B 0,C 180,E1 6451.891,E2 6451.891} C_VEL
LIN {X 0,Y 480.674,Z 702.53,A -85,B 0,C 180,E1 6457.859,E2 6457.859} C_VEL
LIN {X 0,Y 480.891,Z 702.53,A -85,B 0,C 180,E1 6463.584,E2 6463.584} C_VEL
LIN {X 0,Y 480.983,Z 702.53,A -85,B 0,C 180,E1 6469.138,E2 6469.138} C_VEL
LIN {X 0,Y 481.173,Z 702.53,A -85,B 0,C 180,E1 6474.588,E2 6474.588} C_VEL
LIN {X 0,Y 481.27,Z 702.53,A -85,B 0,C 180,E1 6479.986,E2 6479.986} C_VEL
LIN {X 0,Y 481.198,Z 702.53,A -85,B 0,C 180,E1 6485.383,E2 6485.383} C_VEL
LIN {X 0,Y 480.989,Z 702.53,A -85,B 0,C 180,E1 6490.833,E2 6490.833} C_VEL
LIN {X 0,Y 480.861,Z 702.53,A -85,B 0,C 180,E1 6496.387,E2 6496.387} C_VEL
LIN {X 0,Y 480.741,Z 702.53,A -85,B 0,C 180,E1 6502.107,E2 6502.107} C_VEL
LIN {X 0,Y 480.479,Z 702.53,A -85,B 0,C 180,E1 6508.432,E2 6508.432} C_VEL
LIN {X 0,Y 480.45,Z 702.53,A -85,B 0,C 180,E1 6514.4,E2 6514.4} C_VEL
LIN {X 0,Y 480.55,Z 702.53,A -85,B 0,C 180,E1 6518.876,E2 6518.876} C_VEL
LIN {X 0,Y 480.466,Z 702.53,A -85,B 0,C 180,E1 6523.75,E2 6523.75} C_VEL
LIN {X 0,Y 480.38,Z 702.53,A -85,B 0,C 180,E1 6528.893,E2 6528.893} C_VEL
LIN {X 0,Y 480.483,Z 702.53,A -85,B 0,C 180,E1 6534.698,E2 6534.698} C_VEL
LIN {X 0,Y 480.613,Z 702.53,A -85,B 0,C 180,E1 6539.844,E2 6539.844} C_VEL
LIN {X 0,Y 480.658,Z 702.53,A -85,B 0,C 180,E1 6545.912,E2 6545.912} C_VEL
LIN {X 0,Y 480.8,Z 702.53,A -85,B 0,C 180,E1 6551.708,E2 6551.708} C_VEL
LIN {X 0,Y 480.956,Z 702.53,A -85,B 0,C 180,E1 6557.313,E2 6557.313} C_VEL
LIN {X 0,Y 481.08,Z 702.53,A -85,B 0,C 180,E1 6562.792,E2 6562.792} C_VEL
LIN {X 0,Y 481.108,Z 702.53,A -85,B 0,C 180,E1 6564.432,E2 6564.432} C_VEL
LIN {X 0,Y 495.913,Z 740.048,A -85,B 0,C 180,E1 6566.571,E2 6566.571} C_VEL
LIN {X 0,Y 493.771,Z 777.18,A -85,B 0,C 180,E1 6568.184,E2 6568.184} C_VEL
LIN {X 0,Y 491.02,Z 810.249,A -85,B 0,C 180,E1 6570.338,E2 6570.338} C_VEL
LIN {X 0,Y 487.988,Z 841.776,A -85,B 0,C 180,E1 6573.213,E2 6573.213} C_VEL
LIN {X 0,Y 485.456,Z 868.49,A -85,B 0,C 180,E1 6576.57,E2 6576.57} C_VEL
LIN {X 0,Y 483.477,Z 890.516,A -85,B 0,C 180,E1 6580.306,E2 6580.306} C_VEL
LIN {X 0,Y 482.102,Z 910.269,A -85,B 0,C 180,E1 6584.965,E2 6584.965} C_VEL
LIN {X 0,Y 481.644,Z 922.004,A -85,B 0,C 180,E1 6589.136,E2 6589.136} C_VEL
LIN {X 0,Y 481.241,Z 928.062,A -85,B 0,C 180,E1 6592.737,E2 6592.737} C_VEL
LIN {X 0,Y 481.016,Z 930.335,A -85,B 0,C 180,E1 6596.053,E2 6596.053} C_VEL
LIN {X 0,Y 481.193,Z 929.089,A -85,B 0,C 180,E1 6600.117,E2 6600.117} C_VEL
LIN {X 0,Y 481.633,Z 922.944,A -85,B 0,C 180,E1 6604.331,E2 6604.331} C_VEL
LIN {X 0,Y 482.066,Z 911.613,A -85,B 0,C 180,E1 6608.543,E2 6608.543} C_VEL
LIN {X 0,Y 483.218,Z 893.029,A -85,B 0,C 180,E1 6613.118,E2 6613.118} C_VEL
LIN {X 0,Y 485.23,Z 870.372,A -85,B 0,C 180,E1 6617.088,E2 6617.088} C_VEL
LIN {X 0,Y 487.884,Z 844.17,A -85,B 0,C 180,E1 6620.46,E2 6620.46} C_VEL
LIN {X 0,Y 490.924,Z 813.516,A -85,B 0,C 180,E1 6623.355,E2 6623.355} C_VEL
LIN {X 0,Y 493.789,Z 780.107,A -85,B 0,C 180,E1 6625.602,E2 6625.602} C_VEL
LIN {X 0,Y 496.103,Z 745.073,A -85,B 0,C 180,E1 6627.182,E2 6627.182} C_VEL
LIN {X 0,Y 495.477,Z 737.954,A -85,B 0,C 180,E1 6627.495,E2 6627.495} C_VEL
LIN {X 0,Y 480.626,Z 702.53,A -85,B 0,C 180,E1 6629.601,E2 6629.601} C_VEL
LIN {X 0,Y 480.681,Z 702.53,A -85,B 0,C 180,E1 6635.935,E2 6635.935} C_VEL
LIN {X 0,Y 480.895,Z 702.53,A -85,B 0,C 180,E1 6641.732,E2 6641.732} C_VEL
LIN {X 0,Y 481.042,Z 702.53,A -85,B 0,C 180,E1 6647.333,E2 6647.333} C_VEL
LIN {X 0,Y 481.068,Z 702.53,A -85,B 0,C 180,E1 6652.808,E2 6652.808} C_VEL
LIN {X 0,Y 481.171,Z 702.53,A -85,B 0,C 180,E1 6658.218,E2 6658.218} C_VEL
LIN {X 0,Y 481.205,Z 702.53,A -85,B 0,C 180,E1 6663.609,E2 6663.609} C_VEL
LIN {X 0,Y 481.002,Z 702.53,A -85,B 0,C 180,E1 6669.037,E2 6669.037} C_VEL
LIN {X 0,Y 480.85,Z 702.53,A -85,B 0,C 180,E1 6674.552,E2 6674.552} C_VEL
LIN {X 0,Y 480.736,Z 702.53,A -85,B 0,C 180,E1 6680.21,E2 6680.21} C_VEL
LIN {X 0,Y 480.613,Z 702.53,A -85,B 0,C 180,E1 6686.086,E2 6686.086} C_VEL
LIN {X 0,Y 480.442,Z 702.53,A -85,B 0,C 180,E1 6692.281,E2 6692.281} C_VEL
LIN {X 0,Y 480.529,Z 702.53,A -85,B 0,C 180,E1 6698.915,E2 6698.915} C_VEL
LIN {X 0,Y 480.419,Z 702.53,A -85,B 0,C 180,E1 6703.743,E2 6703.743} C_VEL
LIN {X 0,Y 480.301,Z 702.53,A -85,B 0,C 180,E1 6709.715,E2 6709.715} C_VEL
LIN {X 0,Y 480.428,Z 702.53,A -85,B 0,C 180,E1 6711.649,E2 6711.649} C_VEL
LIN {X 0,Y 483.832,Z 707.561,A -85,B 0,C 180,E1 6712.097,E2 6712.097} C_VEL
LIN {X 0,Y 487.022,Z 732.872,A -85,B 0,C 180,E1 6712.795,E2 6712.795} C_VEL
LIN {X 0,Y 487.924,Z 735.054,A -85,B 0,C 180,E1 6712.911,E2 6712.911} C_VEL
LIN {X 0,Y 494.236,Z 747.481,A -85,B 0,C 180,E1 6713.613,E2 6713.613} C_VEL
LIN {X 0,Y 492.798,Z 789.604,A -85,B 0,C 180,E1 6714.624,E2 6714.624} C_VEL
LIN {X 0,Y 490.134,Z 828.97,A -85,B 0,C 180,E1 6716.28,E2 6716.28} C_VEL
LIN {X 0,Y 486.726,Z 866.206,A -85,B 0,C 180,E1 6718.588,E2 6718.588} C_VEL
LIN {X 0,Y 483.295,Z 899.634,A -85,B 0,C 180,E1 6721.43,E2 6721.43} C_VEL
LIN {X 0,Y 479.906,Z 929.36,A -85,B 0,C 180,E1 6724.881,E2 6724.881} C_VEL
LIN {X 0,Y 477.032,Z 955.524,A -85,B 0,C 180,E1 6728.88,E2 6728.88} C_VEL
LIN {X 0,Y 475.095,Z 976.245,A -85,B 0,C 180,E1 6733.085,E2 6733.085} C_VEL
LIN {X 0,Y 474.052,Z 992.4,A -85,B 0,C 180,E1 6737.592,E2 6737.592} C_VEL
LIN {X 0,Y 473.685,Z 1002.665,A -85,B 0,C 180,E1 6741.792,E2 6741.792} C_VEL
LIN {X 0,Y 473.523,Z 1008.908,A -85,B 0,C 180,E1 6746.345,E2 6746.345} C_VEL
LIN {X 0,Y 473.539,Z 1010.5,A -85,B 0,C 180,E1 6750,E2 6750} C_VEL
LIN {X 0,Y 473.496,Z 1008.911,A -85,B 0,C 180,E1 6753.654,E2 6753.654} C_VEL
LIN {X 0,Y 473.709,Z 1002.628,A -85,B 0,C 180,E1 6758.227,E2 6758.227} C_VEL
LIN {X 0,Y 474.308,Z 989.999,A -85,B 0,C 180,E1 6763.187,E2 6763.187} C_VEL
LIN {X 0,Y 475.518,Z 972.295,A -85,B 0,C 180,E1 6767.813,E2 6767.813} C_VEL
LIN {X 0,Y 477.622,Z 950.199,A -85,B 0,C 180,E1 6772.027,E2 6772.027} C_VEL
LIN {X 0,Y 480.468,Z 923.855,A -85,B 0,C 180,E1 6775.835,E2 6775.835} C_VEL
LIN {X 0,Y 483.955,Z 893.308,A -85,B 0,C 180,E1 6779.177,E2 6779.177} C_VEL
LIN {X 0,Y 487.364,Z 859.664,A -85,B 0,C 180,E1 6781.891,E2 6781.891} C_VEL
LIN {X 0,Y 490.608,Z 822.92,A -85,B 0,C 180,E1 6784.047,E2 6784.047} C_VEL
LIN {X 0,Y 493.218,Z 783.451,A -85,B 0,C 180,E1 6785.588,E2 6785.588} C_VEL
LIN {X 0,Y 494.062,Z 747.292,A -85,B 0,C 180,E1 6786.439,E2 6786.439} C_VEL
LIN {X 0,Y 472.596,Z 702.53,A -85,B 0,C 180,E1 6789.13,E2 6789.13} C_VEL
LIN {X 0,Y 472.47,Z 702.53,A -85,B 0,C 180,E1 6795.352,E2 6795.352} C_VEL
LIN {X 0,Y 472.414,Z 702.53,A -85,B 0,C 180,E1 6800.286,E2 6800.286} C_VEL
LIN {X 0,Y 472.572,Z 702.53,A -85,B 0,C 180,E1 6806.123,E2 6806.123} C_VEL
LIN {X 0,Y 472.677,Z 702.53,A -85,B 0,C 180,E1 6811.379,E2 6811.379} C_VEL
LIN {X 0,Y 472.761,Z 702.53,A -85,B 0,C 180,E1 6817.768,E2 6817.768} C_VEL
LIN {X 0,Y 472.947,Z 702.53,A -85,B 0,C 180,E1 6823.301,E2 6823.301} C_VEL
LIN {X 0,Y 473.061,Z 702.53,A -85,B 0,C 180,E1 6828.954,E2 6828.954} C_VEL
LIN {X 0,Y 473.257,Z 702.53,A -85,B 0,C 180,E1 6834.497,E2 6834.497} C_VEL
LIN {X 0,Y 473.37,Z 702.53,A -85,B 0,C 180,E1 6839.985,E2 6839.985} C_VEL
LIN {X 0,Y 473.284,Z 702.53,A -85,B 0,C 180,E1 6845.473,E2 6845.473} C_VEL
LIN {X 0,Y 473.084,Z 702.53,A -85,B 0,C 180,E1 6851.016,E2 6851.016} C_VEL
LIN {X 0,Y 472.901,Z 702.53,A -85,B 0,C 180,E1 6856.805,E2 6856.805} C_VEL
LIN {X 0,Y 472.779,Z 702.53,A -85,B 0,C 180,E1 6862.499,E2 6862.499} C_VEL
LIN {X 0,Y 472.591,Z 702.53,A -85,B 0,C 180,E1 6868.594,E2 6868.594} C_VEL
LIN {X 0,Y 472.576,Z 702.53,A -85,B 0,C 180,E1 6875.056,E2 6875.056} C_VEL
LIN {X 0,Y 472.551,Z 702.53,A -85,B 0,C 180,E1 6879.968,E2 6879.968} C_VEL
LIN {X 0,Y 472.449,Z 702.53,A -85,B 0,C 180,E1 6885.357,E2 6885.357} C_VEL
LIN {X 0,Y 472.443,Z 702.53,A -85,B 0,C 180,E1 6890.297,E2 6890.297} C_VEL
LIN {X 0,Y 472.578,Z 702.53,A -85,B 0,C 180,E1 6896.075,E2 6896.075} C_VEL
LIN {X 0,Y 472.671,Z 702.53,A -85,B 0,C 180,E1 6901.388,E2 6901.388} C_VEL
LIN {X 0,Y 472.841,Z 702.53,A -85,B 0,C 180,E1 6907.673,E2 6907.673} C_VEL
LIN {X 0,Y 472.931,Z 702.53,A -85,B 0,C 180,E1 6913.312,E2 6913.312} C_VEL
LIN {X 0,Y 473.087,Z 702.53,A -85,B 0,C 180,E1 6918.967,E2 6918.967} C_VEL
LIN {X 0,Y 473.183,Z 702.53,A -85,B 0,C 180,E1 6923.764,E2 6923.764} C_VEL
LIN {X 0,Y 488.236,Z 739.656,A -85,B 0,C 180,E1 6925.983,E2 6925.983} C_VEL
LIN {X 0,Y 488.957,Z 747.793,A -85,B 0,C 180,E1 6926.36,E2 6926.36} C_VEL
LIN {X 0,Y 486.407,Z 784.645,A -85,B 0,C 180,E1 6928.111,E2 6928.111} C_VEL
LIN {X 0,Y 483.198,Z 818.82,A -85,B 0,C 180,E1 6930.559,E2 6930.559} C_VEL
LIN {X 0,Y 480.069,Z 849.216,A -85,B 0,C 180,E1 6933.605,E2 6933.605} C_VEL
LIN {X 0,Y 477.246,Z 875.883,A -85,B 0,C 180,E1 6937.266,E2 6937.266} C_VEL
LIN {X 0,Y 475.277,Z 896.812,A -85,B 0,C 180,E1 6941.214,E2 6941.214} C_VEL
LIN {X 0,Y 474.189,Z 912.03,A -85,B 0,C 180,E1 6945.221,E2 6945.221} C_VEL
LIN {X 0,Y 473.696,Z 923.993,A -85,B 0,C 180,E1 6949.968,E2 6949.968} C_VEL
LIN {X 0,Y 473.156,Z 929.657,A -85,B 0,C 180,E1 6954.495,E2 6954.495} C_VEL
LIN {X 0,Y 473.137,Z 930.122,A -85,B 0,C 180,E1 6958.582,E2 6958.582} C_VEL
LIN {X 0,Y 473.601,Z 925.941,A -85,B 0,C 180,E1 6962.798,E2 6962.798} C_VEL
LIN {X 0,Y 473.998,Z 916.115,A -85,B 0,C 180,E1 6967.301,E2 6967.301} C_VEL
LIN {X 0,Y 474.891,Z 902.269,A -85,B 0,C 180,E1 6971.432,E2 6971.432} C_VEL
LIN {X 0,Y 476.671,Z 882.95,A -85,B 0,C 180,E1 6975.477,E2 6975.477} C_VEL
LIN {X 0,Y 479.224,Z 858.126,A -85,B 0,C 180,E1 6979.25,E2 6979.25} C_VEL
LIN {X 0,Y 482.195,Z 830.415,A -85,B 0,C 180,E1 6982.349,E2 6982.349} C_VEL
LIN {X 0,Y 485.326,Z 799.137,A -85,B 0,C 180,E1 6984.915,E2 6984.915} C_VEL
LIN {X 0,Y 488.181,Z 764.575,A -85,B 0,C 180,E1 6986.902,E2 6986.902} C_VEL
LIN {X 0,Y 489.06,Z 741.253,A -85,B 0,C 180,E1 6987.875,E2 6987.875} C_VEL
LIN {X 0,Y 474.284,Z 707.29,A -85,B 0,C 180,E1 6990.045,E2 6990.045} C_VEL
LIN {X 0,Y 472.652,Z 702.53,A -85,B 0,C 180,E1 6990.364,E2 6990.364} C_VEL
LIN {X 0,Y 472.764,Z 702.53,A -85,B 0,C 180,E1 6995.506,E2 6995.506} C_VEL
LIN {X 0,Y 472.963,Z 702.53,A -85,B 0,C 180,E1 7001.414,E2 7001.414} C_VEL
LIN {X 0,Y 473.146,Z 702.53,A -85,B 0,C 180,E1 7007.118,E2 7007.118} C_VEL
LIN {X 0,Y 473.155,Z 702.53,A -85,B 0,C 180,E1 7012.687,E2 7012.687} C_VEL
LIN {X 0,Y 473.269,Z 702.53,A -85,B 0,C 180,E1 7018.188,E2 7018.188} C_VEL
LIN {X 0,Y 473.296,Z 702.53,A -85,B 0,C 180,E1 7023.67,E2 7023.67} C_VEL
LIN {X 0,Y 473.086,Z 702.53,A -85,B 0,C 180,E1 7029.19,E2 7029.19} C_VEL
LIN {X 0,Y 472.916,Z 702.53,A -85,B 0,C 180,E1 7034.801,E2 7034.801} C_VEL
LIN {X 0,Y 472.785,Z 702.53,A -85,B 0,C 180,E1 7040.565,E2 7040.565} C_VEL
LIN {X 0,Y 472.626,Z 702.53,A -85,B 0,C 180,E1 7046.619,E2 7046.619} C_VEL
LIN {X 0,Y 472.47,Z 702.53,A -85,B 0,C 180,E1 7052.894,E2 7052.894} C_VEL
LIN {X 0,Y 472.62,Z 702.53,A -85,B 0,C 180,E1 7057.356,E2 7057.356} C_VEL
LIN {X 0,Y 472.465,Z 702.53,A -85,B 0,C 180,E1 7062.726,E2 7062.726} C_VEL
LIN {X 0,Y 472.383,Z 702.53,A -85,B 0,C 180,E1 7067.867,E2 7067.867} C_VEL
LIN {X 0,Y 472.475,Z 702.53,A -85,B 0,C 180,E1 7071.044,E2 7071.044} C_VEL
LIN {X 0,Y 487.924,Z 735.054,A -85,B 0,C 180,E1 7072.911,E2 7072.911} C_VEL
LIN {X 0,Y 489.403,Z 743.308,A -85,B 0,C 180,E1 7073.167,E2 7073.167} C_VEL
LIN {X 0,Y 487.537,Z 758.497,A -85,B 0,C 180,E1 7073.317,E2 7073.317} C_VEL
LIN {X 0,Y 485.371,Z 799.581,A -85,B 0,C 180,E1 7074.479,E2 7074.479} C_VEL
LIN {X 0,Y 482.116,Z 840.596,A -85,B 0,C 180,E1 7076.456,E2 7076.456} C_VEL
LIN {X 0,Y 478.481,Z 876.889,A -85,B 0,C 180,E1 7078.995,E2 7078.995} C_VEL
LIN {X 0,Y 474.679,Z 910.758,A -85,B 0,C 180,E1 7082.21,E2 7082.21} C_VEL
LIN {X 0,Y 471.547,Z 937.615,A -85,B 0,C 180,E1 7085.621,E2 7085.621} C_VEL
LIN {X 0,Y 468.753,Z 962.137,A -85,B 0,C 180,E1 7089.753,E2 7089.753} C_VEL
LIN {X 0,Y 467.001,Z 981.287,A -85,B 0,C 180,E1 7094.058,E2 7094.058} C_VEL
LIN {X 0,Y 466.095,Z 996.305,A -85,B 0,C 180,E1 7098.799,E2 7098.799} C_VEL
LIN {X 0,Y 465.751,Z 1005.749,A -85,B 0,C 180,E1 7103.488,E2 7103.488} C_VEL
LIN {X 0,Y 465.641,Z 1010.089,A -85,B 0,C 180,E1 7108.143,E2 7108.143} C_VEL
LIN {X 0,Y 465.693,Z 1010.09,A -85,B 0,C 180,E1 7111.857,E2 7111.857} C_VEL
LIN {X 0,Y 465.743,Z 1005.754,A -85,B 0,C 180,E1 7116.511,E2 7116.511} C_VEL
LIN {X 0,Y 466.026,Z 996.306,A -85,B 0,C 180,E1 7121.203,E2 7121.203} C_VEL
LIN {X 0,Y 467.06,Z 981.291,A -85,B 0,C 180,E1 7125.94,E2 7125.94} C_VEL
LIN {X 0,Y 469.057,Z 959.651,A -85,B 0,C 180,E1 7130.725,E2 7130.725} C_VEL
LIN {X 0,Y 471.935,Z 934.602,A -85,B 0,C 180,E1 7134.814,E2 7134.814} C_VEL
LIN {X 0,Y 475.273,Z 905.874,A -85,B 0,C 180,E1 7138.327,E2 7138.327} C_VEL
LIN {X 0,Y 479.138,Z 870.863,A -85,B 0,C 180,E1 7141.507,E2 7141.507} C_VEL
LIN {X 0,Y 482.817,Z 834.404,A -85,B 0,C 180,E1 7143.922,E2 7143.922} C_VEL
LIN {X 0,Y 485.691,Z 797.322,A -85,B 0,C 180,E1 7145.63,E2 7145.63} C_VEL
LIN {X 0,Y 487.874,Z 757.358,A -85,B 0,C 180,E1 7146.726,E2 7146.726} C_VEL
LIN {X 0,Y 487.15,Z 749.302,A -85,B 0,C 180,E1 7146.95,E2 7146.95} C_VEL
LIN {X 0,Y 464.762,Z 703.866,A -85,B 0,C 180,E1 7149.716,E2 7149.716} C_VEL
LIN {X 0,Y 464.645,Z 702.53,A -85,B 0,C 180,E1 7149.85,E2 7149.85} C_VEL
LIN {X 0,Y 464.541,Z 702.53,A -85,B 0,C 180,E1 7155.614,E2 7155.614} C_VEL
LIN {X 0,Y 464.474,Z 702.53,A -85,B 0,C 180,E1 7161.873,E2 7161.873} C_VEL
LIN {X 0,Y 464.654,Z 702.53,A -85,B 0,C 180,E1 7167.606,E2 7167.606} C_VEL
LIN {X 0,Y 464.75,Z 702.53,A -85,B 0,C 180,E1 7172.953,E2 7172.953} C_VEL
LIN {X 0,Y 464.885,Z 702.53,A -85,B 0,C 180,E1 7179.069,E2 7179.069} C_VEL
LIN {X 0,Y 465.087,Z 702.53,A -85,B 0,C 180,E1 7184.944,E2 7184.944} C_VEL
LIN {X 0,Y 465.243,Z 702.53,A -85,B 0,C 180,E1 7190.654,E2 7190.654} C_VEL
LIN {X 0,Y 465.496,Z 702.53,A -85,B 0,C 180,E1 7196.269,E2 7196.269} C_VEL
LIN {X 0,Y 465.614,Z 702.53,A -85,B 0,C 180,E1 7201.842,E2 7201.842} C_VEL
LIN {X 0,Y 465.317,Z 702.53,A -85,B 0,C 180,E1 7207.437,E2 7207.437} C_VEL
LIN {X 0,Y 465.114,Z 702.53,A -85,B 0,C 180,E1 7213.264,E2 7213.264} C_VEL
LIN {X 0,Y 464.893,Z 702.53,A -85,B 0,C 180,E1 7219.725,E2 7219.725} C_VEL
LIN {X 0,Y 464.789,Z 702.53,A -85,B 0,C 180,E1 7224.943,E2 7224.943} C_VEL
LIN {X 0,Y 464.572,Z 702.53,A -85,B 0,C 180,E1 7231.287,E2 7231.287} C_VEL
LIN {X 0,Y 464.664,Z 702.53,A -85,B 0,C 180,E1 7235.744,E2 7235.744} C_VEL
LIN {X 0,Y 464.576,Z 702.53,A -85,B 0,C 180,E1 7241.662,E2 7241.662} C_VEL
LIN {X 0,Y 464.475,Z 702.53,A -85,B 0,C 180,E1 7248.314,E2 7248.314} C_VEL
LIN {X 0,Y 464.623,Z 702.53,A -85,B 0,C 180,E1 7254.243,E2 7254.243} C_VEL
LIN {X 0,Y 464.726,Z 702.53,A -85,B 0,C 180,E1 7260.852,E2 7260.852} C_VEL
LIN {X 0,Y 464.842,Z 702.53,A -85,B 0,C 180,E1 7267.073,E2 7267.073} C_VEL
LIN {X 0,Y 465.006,Z 702.53,A -85,B 0,C 180,E1 7273.019,E2 7273.019} C_VEL
LIN {X 0,Y 465.161,Z 702.53,A -85,B 0,C 180,E1 7278.776,E2 7278.776} C_VEL
LIN {X 0,Y 465.264,Z 702.53,A -85,B 0,C 180,E1 7283.073,E2 7283.073} C_VEL
LIN {X 0,Y 480.993,Z 740.42,A -85,B 0,C 180,E1 7285.447,E2 7285.447} C_VEL
LIN {X 0,Y 482.251,Z 748.81,A -85,B 0,C 180,E1 7285.887,E2 7285.887} C_VEL
LIN {X 0,Y 479.553,Z 785.066,A -85,B 0,C 180,E1 7287.633,E2 7287.633} C_VEL
LIN {X 0,Y 476.161,Z 819.342,A -85,B 0,C 180,E1 7290.119,E2 7290.119} C_VEL
LIN {X 0,Y 472.825,Z 849.723,A -85,B 0,C 180,E1 7293.202,E2 7293.202} C_VEL
LIN {X 0,Y 469.847,Z 875.963,A -85,B 0,C 180,E1 7296.839,E2 7296.839} C_VEL
LIN {X 0,Y 467.761,Z 896.607,A -85,B 0,C 180,E1 7300.751,E2 7300.751} C_VEL
LIN {X 0,Y 466.422,Z 912.65,A -85,B 0,C 180,E1 7305.001,E2 7305.001} C_VEL
LIN {X 0,Y 465.87,Z 923.779,A -85,B 0,C 180,E1 7309.507,E2 7309.507} C_VEL
LIN {X 0,Y 465.409,Z 928.637,A -85,B 0,C 180,E1 7312.898,E2 7312.898} C_VEL
LIN {X 0,Y 465.154,Z 930.69,A -85,B 0,C 180,E1 7317.012,E2 7317.012} C_VEL
LIN {X 0,Y 465.48,Z 928.433,A -85,B 0,C 180,E1 7321.245,E2 7321.245} C_VEL
LIN {X 0,Y 466.003,Z 921.314,A -85,B 0,C 180,E1 7325.654,E2 7325.654} C_VEL
LIN {X 0,Y 466.757,Z 908.203,A -85,B 0,C 180,E1 7330.286,E2 7330.286} C_VEL
LIN {X 0,Y 468.379,Z 890.626,A -85,B 0,C 180,E1 7334.468,E2 7334.468} C_VEL
LIN {X 0,Y 471.029,Z 866.704,A -85,B 0,C 180,E1 7338.539,E2 7338.539} C_VEL
LIN {X 0,Y 473.992,Z 840.552,A -85,B 0,C 180,E1 7341.807,E2 7341.807} C_VEL
LIN {X 0,Y 477.47,Z 809.275,A -85,B 0,C 180,E1 7344.677,E2 7344.677} C_VEL
LIN {X 0,Y 480.695,Z 775.906,A -85,B 0,C 180,E1 7346.847,E2 7346.847} C_VEL
LIN {X 0,Y 482.321,Z 743.673,A -85,B 0,C 180,E1 7348.313,E2 7348.313} C_VEL
LIN {X 0,Y 468.02,Z 710.712,A -85,B 0,C 180,E1 7350.524,E2 7350.524} C_VEL
LIN {X 0,Y 464.769,Z 702.53,A -85,B 0,C 180,E1 7351,E2 7351} C_VEL
LIN {X 0,Y 464.871,Z 702.53,A -85,B 0,C 180,E1 7357.096,E2 7357.096} C_VEL
LIN {X 0,Y 465.119,Z 702.53,A -85,B 0,C 180,E1 7363.042,E2 7363.042} C_VEL
LIN {X 0,Y 465.197,Z 702.53,A -85,B 0,C 180,E1 7368.795,E2 7368.795} C_VEL
LIN {X 0,Y 465.345,Z 702.53,A -85,B 0,C 180,E1 7374.434,E2 7374.434} C_VEL
LIN {X 0,Y 465.506,Z 702.53,A -85,B 0,C 180,E1 7380.015,E2 7380.015} C_VEL
LIN {X 0,Y 465.37,Z 702.53,A -85,B 0,C 180,E1 7385.596,E2 7385.596} C_VEL
LIN {X 0,Y 465.104,Z 702.53,A -85,B 0,C 180,E1 7391.238,E2 7391.238} C_VEL
LIN {X 0,Y 464.976,Z 702.53,A -85,B 0,C 180,E1 7396.994,E2 7396.994} C_VEL
LIN {X 0,Y 464.777,Z 702.53,A -85,B 0,C 180,E1 7402.941,E2 7402.941} C_VEL
LIN {X 0,Y 464.63,Z 702.53,A -85,B 0,C 180,E1 7409.164,E2 7409.164} C_VEL
LIN {X 0,Y 464.635,Z 702.53,A -85,B 0,C 180,E1 7415.783,E2 7415.783} C_VEL
LIN {X 0,Y 464.547,Z 702.53,A -85,B 0,C 180,E1 7421.658,E2 7421.658} C_VEL
LIN {X 0,Y 464.44,Z 702.53,A -85,B 0,C 180,E1 7428.364,E2 7428.364} C_VEL
LIN {X 0,Y 464.522,Z 702.53,A -85,B 0,C 180,E1 7430.304,E2 7430.304} C_VEL
LIN {X 0,Y 484.424,Z 743.726,A -85,B 0,C 180,E1 7432.783,E2 7432.783} C_VEL
LIN {X 0,Y 487.645,Z 751.849,A -85,B 0,C 180,E1 7433.189,E2 7433.189} C_VEL
LIN {X 0,Y 487.537,Z 758.497,A -85,B 0,C 180,E1 7433.317,E2 7433.317} C_VEL
LIN {X 0,Y 483.556,Z 775.556,A -85,B 0,C 180,E1 7433.453,E2 7433.453} C_VEL
LIN {X 0,Y 479.2,Z 792.348,A -85,B 0,C 180,E1 7433.725,E2 7433.725} C_VEL
LIN {X 0,Y 476.245,Z 829.713,A -85,B 0,C 180,E1 7435.375,E2 7435.375} C_VEL
LIN {X 0,Y 472.471,Z 866.322,A -85,B 0,C 180,E1 7437.731,E2 7437.731} C_VEL
LIN {X 0,Y 468.554,Z 899.966,A -85,B 0,C 180,E1 7440.697,E2 7440.697} C_VEL
LIN {X 0,Y 464.887,Z 930.547,A -85,B 0,C 180,E1 7444.268,E2 7444.268} C_VEL
LIN {X 0,Y 462.065,Z 954.361,A -85,B 0,C 180,E1 7447.94,E2 7447.94} C_VEL
LIN {X 0,Y 459.695,Z 976.097,A -85,B 0,C 180,E1 7452.464,E2 7452.464} C_VEL
LIN {X 0,Y 458.394,Z 992.4,A -85,B 0,C 180,E1 7457.161,E2 7457.161} C_VEL
LIN {X 0,Y 457.949,Z 1002.316,A -85,B 0,C 180,E1 7461.334,E2 7461.334} C_VEL
LIN {X 0,Y 457.734,Z 1008.908,A -85,B 0,C 180,E1 7466.219,E2 7466.219} C_VEL
LIN {X 0,Y 457.753,Z 1010.5,A -85,B 0,C 180,E1 7470,E2 7470} C_VEL
LIN {X 0,Y 457.717,Z 1008.911,A -85,B 0,C 180,E1 7473.78,E2 7473.78} C_VEL
LIN {X 0,Y 457.97,Z 1002.284,A -85,B 0,C 180,E1 7478.683,E2 7478.683} C_VEL
LIN {X 0,Y 458.559,Z 991.041,A -85,B 0,C 180,E1 7483.318,E2 7483.318} C_VEL
LIN {X 0,Y 459.947,Z 973.94,A -85,B 0,C 180,E1 7488.06,E2 7488.06} C_VEL
LIN {X 0,Y 462.434,Z 951.601,A -85,B 0,C 180,E1 7492.546,E2 7492.546} C_VEL
LIN {X 0,Y 465.574,Z 925.047,A -85,B 0,C 180,E1 7496.466,E2 7496.466} C_VEL
LIN {X 0,Y 469.476,Z 892.877,A -85,B 0,C 180,E1 7500.03,E2 7500.03} C_VEL
LIN {X 0,Y 473.547,Z 857.894,A -85,B 0,C 180,E1 7502.918,E2 7502.918} C_VEL
LIN {X 0,Y 477.154,Z 821.478,A -85,B 0,C 180,E1 7505.091,E2 7505.091} C_VEL
LIN {X 0,Y 480.013,Z 783.11,A -85,B 0,C 180,E1 7506.618,E2 7506.618} C_VEL
LIN {X 0,Y 480.777,Z 752.32,A -85,B 0,C 180,E1 7507.407,E2 7507.407} C_VEL
LIN {X 0,Y 456.8,Z 703.824,A -85,B 0,C 180,E1 7510.473,E2 7510.473} C_VEL
LIN {X 0,Y 456.676,Z 702.53,A -85,B 0,C 180,E1 7510.528,E2 7510.528} C_VEL
LIN {X 0,Y 456.624,Z 702.53,A -85,B 0,C 180,E1 7516.639,E2 7516.639} C_VEL
LIN {X 0,Y 456.589,Z 702.53,A -85,B 0,C 180,E1 7523.486,E2 7523.486} C_VEL
LIN {X 0,Y 456.758,Z 702.53,A -85,B 0,C 180,E1 7530.283,E2 7530.283} C_VEL
LIN {X 0,Y 456.848,Z 702.53,A -85,B 0,C 180,E1 7536.638,E2 7536.638} C_VEL
LIN {X 0,Y 457.117,Z 702.53,A -85,B 0,C 180,E1 7543.204,E2 7543.204} C_VEL
LIN {X 0,Y 457.232,Z 702.53,A -85,B 0,C 180,E1 7548.566,E2 7548.566} C_VEL
LIN {X 0,Y 457.447,Z 702.53,A -85,B 0,C 180,E1 7554.307,E2 7554.307} C_VEL
LIN {X 0,Y 457.599,Z 702.53,A -85,B 0,C 180,E1 7559.985,E2 7559.985} C_VEL
LIN {X 0,Y 457.473,Z 702.53,A -85,B 0,C 180,E1 7565.663,E2 7565.663} C_VEL
LIN {X 0,Y 457.241,Z 702.53,A -85,B 0,C 180,E1 7571.403,E2 7571.403} C_VEL
LIN {X 0,Y 457.051,Z 702.53,A -85,B 0,C 180,E1 7577.266,E2 7577.266} C_VEL
LIN {X 0,Y 456.889,Z 702.53,A -85,B 0,C 180,E1 7583.327,E2 7583.327} C_VEL
LIN {X 0,Y 456.669,Z 702.53,A -85,B 0,C 180,E1 7589.688,E2 7589.688} C_VEL
LIN {X 0,Y 456.664,Z 702.53,A -85,B 0,C 180,E1 7596.47,E2 7596.47} C_VEL
LIN {X 0,Y 456.691,Z 702.53,A -85,B 0,C 180,E1 7601.333,E2 7601.333} C_VEL
LIN {X 0,Y 456.616,Z 702.53,A -85,B 0,C 180,E1 7606.604,E2 7606.604} C_VEL
LIN {X 0,Y 456.616,Z 702.53,A -85,B 0,C 180,E1 7613.497,E2 7613.497} C_VEL
LIN {X 0,Y 456.75,Z 702.53,A -85,B 0,C 180,E1 7620.293,E2 7620.293} C_VEL
LIN {X 0,Y 456.92,Z 702.53,A -85,B 0,C 180,E1 7626.652,E2 7626.652} C_VEL
LIN {X 0,Y 457.099,Z 702.53,A -85,B 0,C 180,E1 7633.114,E2 7633.114} C_VEL
LIN {X 0,Y 457.233,Z 702.53,A -85,B 0,C 180,E1 7638.579,E2 7638.579} C_VEL
LIN {X 0,Y 457.402,Z 703.297,A -85,B 0,C 180,E1 7642.417,E2 7642.417} C_VEL
LIN {X 0,Y 473.394,Z 739.897,A -85,B 0,C 180,E1 7644.817,E2 7644.817} C_VEL
LIN {X 0,Y 475.593,Z 749.599,A -85,B 0,C 180,E1 7645.394,E2 7645.394} C_VEL
LIN {X 0,Y 472.778,Z 785.432,A -85,B 0,C 180,E1 7647.142,E2 7647.142} C_VEL
LIN {X 0,Y 469.179,Z 819.731,A -85,B 0,C 180,E1 7649.655,E2 7649.655} C_VEL
LIN {X 0,Y 465.575,Z 850.247,A -85,B 0,C 180,E1 7652.787,E2 7652.787} C_VEL
LIN {X 0,Y 462.307,Z 877.272,A -85,B 0,C 180,E1 7656.607,E2 7656.607} C_VEL
LIN {X 0,Y 459.955,Z 898.745,A -85,B 0,C 180,E1 7660.808,E2 7660.808} C_VEL
LIN {X 0,Y 458.575,Z 914.774,A -85,B 0,C 180,E1 7665.264,E2 7665.264} C_VEL
LIN {X 0,Y 457.997,Z 925.331,A -85,B 0,C 180,E1 7669.857,E2 7669.857} C_VEL
LIN {X 0,Y 457.486,Z 929.765,A -85,B 0,C 180,E1 7673.318,E2 7673.318} C_VEL
LIN {X 0,Y 457.276,Z 931.316,A -85,B 0,C 180,E1 7677.517,E2 7677.517} C_VEL
LIN {X 0,Y 457.694,Z 928.534,A -85,B 0,C 180,E1 7681.839,E2 7681.839} C_VEL
LIN {X 0,Y 458.235,Z 920.792,A -85,B 0,C 180,E1 7686.354,E2 7686.354} C_VEL
LIN {X 0,Y 459.143,Z 907.515,A -85,B 0,C 180,E1 7690.933,E2 7690.933} C_VEL
LIN {X 0,Y 461.188,Z 888.247,A -85,B 0,C 180,E1 7695.395,E2 7695.395} C_VEL
LIN {X 0,Y 464.025,Z 864.386,A -85,B 0,C 180,E1 7699.345,E2 7699.345} C_VEL
LIN {X 0,Y 467.545,Z 835.923,A -85,B 0,C 180,E1 7702.8,E2 7702.8} C_VEL
LIN {X 0,Y 471.334,Z 802.991,A -85,B 0,C 180,E1 7705.666,E2 7705.666} C_VEL
LIN {X 0,Y 474.563,Z 768.972,A -85,B 0,C 180,E1 7707.733,E2 7707.733} C_VEL
LIN {X 0,Y 475.743,Z 746.516,A -85,B 0,C 180,E1 7708.732,E2 7708.732} C_VEL
LIN {X 0,Y 462.384,Z 715.141,A -85,B 0,C 180,E1 7710.935,E2 7710.935} C_VEL
LIN {X 0,Y 456.843,Z 702.53,A -85,B 0,C 180,E1 7711.842,E2 7711.842} C_VEL
LIN {X 0,Y 457.001,Z 702.53,A -85,B 0,C 180,E1 7718.723,E2 7718.723} C_VEL
LIN {X 0,Y 457.247,Z 702.53,A -85,B 0,C 180,E1 7724.711,E2 7724.711} C_VEL
LIN {X 0,Y 457.369,Z 702.53,A -85,B 0,C 180,E1 7730.522,E2 7730.522} C_VEL
LIN {X 0,Y 457.54,Z 702.53,A -85,B 0,C 180,E1 7736.234,E2 7736.234} C_VEL
LIN {X 0,Y 457.712,Z 702.53,A -85,B 0,C 180,E1 7741.904,E2 7741.904} C_VEL
LIN {X 0,Y 457.305,Z 702.53,A -85,B 0,C 180,E1 7748.129,E2 7748.129} C_VEL
LIN {X 0,Y 457.166,Z 702.53,A -85,B 0,C 180,E1 7753.372,E2 7753.372} C_VEL
LIN {X 0,Y 456.977,Z 702.53,A -85,B 0,C 180,E1 7759.293,E2 7759.293} C_VEL
LIN {X 0,Y 456.784,Z 702.53,A -85,B 0,C 180,E1 7765.444,E2 7765.444} C_VEL
LIN {X 0,Y 456.609,Z 702.53,A -85,B 0,C 180,E1 7771.932,E2 7771.932} C_VEL
LIN {X 0,Y 456.691,Z 702.53,A -85,B 0,C 180,E1 7778.897,E2 7778.897} C_VEL
LIN {X 0,Y 456.599,Z 702.53,A -85,B 0,C 180,E1 7783.958,E2 7783.958} C_VEL
LIN {X 0,Y 456.57,Z 702.53,A -85,B 0,C 180,E1 7789.559,E2 7789.559} C_VEL
LIN {X 0,Y 463.012,Z 716.415,A -85,B 0,C 180,E1 7790.453,E2 7790.453} C_VEL
LIN {X 0,Y 480.989,Z 752.683,A -85,B 0,C 180,E1 7792.678,E2 7792.678} C_VEL
LIN {X 0,Y 479.2,Z 792.348,A -85,B 0,C 180,E1 7793.725,E2 7793.725} C_VEL
LIN {X 0,Y 469.871,Z 825.231,A -85,B 0,C 180,E1 7794.637,E2 7794.637} C_VEL
LIN {X 0,Y 465.75,Z 863.274,A -85,B 0,C 180,E1 7797.042,E2 7797.042} C_VEL
LIN {X 0,Y 461.444,Z 898.307,A -85,B 0,C 180,E1 7800.127,E2 7800.127} C_VEL
LIN {X 0,Y 457.611,Z 928.312,A -85,B 0,C 180,E1 7803.639,E2 7803.639} C_VEL
LIN {X 0,Y 454.315,Z 955.36,A -85,B 0,C 180,E1 7807.801,E2 7807.801} C_VEL
LIN {X 0,Y 452.171,Z 974.706,A -85,B 0,C 180,E1 7811.803,E2 7811.803} C_VEL
LIN {X 0,Y 450.69,Z 991.036,A -85,B 0,C 180,E1 7816.445,E2 7816.445} C_VEL
LIN {X 0,Y 450.065,Z 1002.316,A -85,B 0,C 180,E1 7821.181,E2 7821.181} C_VEL
LIN {X 0,Y 449.826,Z 1008.907,A -85,B 0,C 180,E1 7826.153,E2 7826.153} C_VEL
LIN {X 0,Y 449.855,Z 1010.5,A -85,B 0,C 180,E1 7830,E2 7830} C_VEL
LIN {X 0,Y 449.813,Z 1008.911,A -85,B 0,C 180,E1 7833.847,E2 7833.847} C_VEL
LIN {X 0,Y 450.079,Z 1002.284,A -85,B 0,C 180,E1 7838.836,E2 7838.836} C_VEL
LIN {X 0,Y 450.818,Z 989.989,A -85,B 0,C 180,E1 7843.891,E2 7843.891} C_VEL
LIN {X 0,Y 452.301,Z 973.264,A -85,B 0,C 180,E1 7848.534,E2 7848.534} C_VEL
LIN {X 0,Y 454.704,Z 952.627,A -85,B 0,C 180,E1 7852.693,E2 7852.693} C_VEL
LIN {X 0,Y 458.275,Z 923.558,A -85,B 0,C 180,E1 7857.009,E2 7857.009} C_VEL
LIN {X 0,Y 462.308,Z 892.395,A -85,B 0,C 180,E1 7860.501,E2 7860.501} C_VEL
LIN {X 0,Y 466.637,Z 857.069,A -85,B 0,C 180,E1 7863.454,E2 7863.454} C_VEL
LIN {X 0,Y 470.511,Z 820.156,A -85,B 0,C 180,E1 7865.667,E2 7865.667} C_VEL
LIN {X 0,Y 473.516,Z 782.227,A -85,B 0,C 180,E1 7867.176,E2 7867.176} C_VEL
LIN {X 0,Y 474.424,Z 755.266,A -85,B 0,C 180,E1 7867.879,E2 7867.879} C_VEL
LIN {X 0,Y 449.899,Z 706.616,A -85,B 0,C 180,E1 7871.097,E2 7871.097} C_VEL
LIN {X 0,Y 448.771,Z 702.53,A -85,B 0,C 180,E1 7871.322,E2 7871.322} C_VEL
LIN {X 0,Y 448.634,Z 702.53,A -85,B 0,C 180,E1 7877.73,E2 7877.73} C_VEL
LIN {X 0,Y 448.658,Z 702.53,A -85,B 0,C 180,E1 7883.825,E2 7883.825} C_VEL
LIN {X 0,Y 448.829,Z 702.53,A -85,B 0,C 180,E1 7889.704,E2 7889.704} C_VEL
LIN {X 0,Y 448.887,Z 702.53,A -85,B 0,C 180,E1 7896.198,E2 7896.198} C_VEL
LIN {X 0,Y 449.134,Z 702.53,A -85,B 0,C 180,E1 7902.387,E2 7902.387} C_VEL
LIN {X 0,Y 449.309,Z 702.53,A -85,B 0,C 180,E1 7908.362,E2 7908.362} C_VEL
LIN {X 0,Y 449.542,Z 702.53,A -85,B 0,C 180,E1 7914.206,E2 7914.206} C_VEL
LIN {X 0,Y 449.711,Z 702.53,A -85,B 0,C 180,E1 7919.985,E2 7919.985} C_VEL
LIN {X 0,Y 449.585,Z 702.53,A -85,B 0,C 180,E1 7925.762,E2 7925.762} C_VEL
LIN {X 0,Y 449.314,Z 702.53,A -85,B 0,C 180,E1 7931.607,E2 7931.607} C_VEL
LIN {X 0,Y 449.106,Z 702.53,A -85,B 0,C 180,E1 7937.582,E2 7937.582} C_VEL
LIN {X 0,Y 448.924,Z 702.53,A -85,B 0,C 180,E1 7943.766,E2 7943.766} C_VEL
LIN {X 0,Y 448.73,Z 702.53,A -85,B 0,C 180,E1 7950.268,E2 7950.268} C_VEL
LIN {X 0,Y 448.749,Z 702.53,A -85,B 0,C 180,E1 7957.22,E2 7957.22} C_VEL
LIN {X 0,Y 448.709,Z 702.53,A -85,B 0,C 180,E1 7962.28,E2 7962.28} C_VEL
LIN {X 0,Y 448.619,Z 702.53,A -85,B 0,C 180,E1 7967.721,E2 7967.721} C_VEL
LIN {X 0,Y 448.687,Z 702.53,A -85,B 0,C 180,E1 7973.775,E2 7973.775} C_VEL
LIN {X 0,Y 448.819,Z 702.53,A -85,B 0,C 180,E1 7979.713,E2 7979.713} C_VEL
LIN {X 0,Y 448.953,Z 702.53,A -85,B 0,C 180,E1 7986.213,E2 7986.213} C_VEL
LIN {X 0,Y 449.123,Z 702.53,A -85,B 0,C 180,E1 7992.399,E2 7992.399} C_VEL
LIN {X 0,Y 449.307,Z 702.53,A -85,B 0,C 180,E1 7998.375,E2 7998.375} C_VEL
LIN {X 0,Y 449.406,Z 702.53,A -85,B 0,C 180,E1 8001.634,E2 8001.634} C_VEL
LIN {X 0,Y 466.823,Z 742.599,A -85,B 0,C 180,E1 8004.371,E2 8004.371} C_VEL
LIN {X 0,Y 468.82,Z 752.313,A -85,B 0,C 180,E1 8004.956,E2 8004.956} C_VEL
LIN {X 0,Y 465.822,Z 787.611,A -85,B 0,C 180,E1 8006.75,E2 8006.75} C_VEL
LIN {X 0,Y 462.18,Z 820.204,A -85,B 0,C 180,E1 8009.182,E2 8009.182} C_VEL
LIN {X 0,Y 458.358,Z 850.766,A -85,B 0,C 180,E1 8012.359,E2 8012.359} C_VEL
LIN {X 0,Y 454.875,Z 877.788,A -85,B 0,C 180,E1 8016.23,E2 8016.23} C_VEL
LIN {X 0,Y 452.411,Z 898.824,A -85,B 0,C 180,E1 8020.389,E2 8020.389} C_VEL
LIN {X 0,Y 450.874,Z 914.523,A -85,B 0,C 180,E1 8024.748,E2 8024.748} C_VEL
LIN {X 0,Y 450.192,Z 925.79,A -85,B 0,C 180,E1 8029.585,E2 8029.585} C_VEL
LIN {X 0,Y 449.548,Z 930.899,A -85,B 0,C 180,E1 8033.754,E2 8033.754} C_VEL
LIN {X 0,Y 449.404,Z 931.943,A -85,B 0,C 180,E1 8038.041,E2 8038.041} C_VEL
LIN {X 0,Y 450.038,Z 927.792,A -85,B 0,C 180,E1 8043.091,E2 8043.091} C_VEL
LIN {X 0,Y 450.652,Z 918.323,A -85,B 0,C 180,E1 8047.85,E2 8047.85} C_VEL
LIN {X 0,Y 451.959,Z 903.886,A -85,B 0,C 180,E1 8052.356,E2 8052.356} C_VEL
LIN {X 0,Y 454.238,Z 884.414,A -85,B 0,C 180,E1 8056.598,E2 8056.598} C_VEL
LIN {X 0,Y 457.4,Z 859.874,A -85,B 0,C 180,E1 8060.47,E2 8060.47} C_VEL
LIN {X 0,Y 461.132,Z 831.049,A -85,B 0,C 180,E1 8063.807,E2 8063.807} C_VEL
LIN {X 0,Y 465.072,Z 798.23,A -85,B 0,C 180,E1 8066.55,E2 8066.55} C_VEL
LIN {X 0,Y 468.574,Z 761.719,A -85,B 0,C 180,E1 8068.626,E2 8068.626} C_VEL
LIN {X 0,Y 468.9,Z 748.381,A -85,B 0,C 180,E1 8069.235,E2 8069.235} C_VEL
LIN {X 0,Y 455.295,Z 716.525,A -85,B 0,C 180,E1 8071.571,E2 8071.571} C_VEL
LIN {X 0,Y 448.926,Z 702.53,A -85,B 0,C 180,E1 8072.585,E2 8072.585} C_VEL
LIN {X 0,Y 449.062,Z 702.53,A -85,B 0,C 180,E1 8078.328,E2 8078.328} C_VEL
LIN {X 0,Y 449.339,Z 702.53,A -85,B 0,C 180,E1 8084.435,E2 8084.435} C_VEL
LIN {X 0,Y 449.441,Z 702.53,A -85,B 0,C 180,E1 8090.354,E2 8090.354} C_VEL
LIN {X 0,Y 449.626,Z 702.53,A -85,B 0,C 180,E1 8096.168,E2 8096.168} C_VEL
LIN {X 0,Y 449.827,Z 702.53,A -85,B 0,C 180,E1 8101.937,E2 8101.937} C_VEL
LIN {X 0,Y 449.452,Z 702.53,A -85,B 0,C 180,E1 8107.732,E2 8107.732} C_VEL
LIN {X 0,Y 449.245,Z 702.53,A -85,B 0,C 180,E1 8113.612,E2 8113.612} C_VEL
LIN {X 0,Y 449.019,Z 702.53,A -85,B 0,C 180,E1 8119.779,E2 8119.779} C_VEL
LIN {X 0,Y 448.873,Z 702.53,A -85,B 0,C 180,E1 8125.925,E2 8125.925} C_VEL
LIN {X 0,Y 448.648,Z 702.53,A -85,B 0,C 180,E1 8132.767,E2 8132.767} C_VEL
LIN {X 0,Y 448.763,Z 702.53,A -85,B 0,C 180,E1 8139.339,E2 8139.339} C_VEL
LIN {X 0,Y 448.61,Z 702.53,A -85,B 0,C 180,E1 8145.057,E2 8145.057} C_VEL
LIN {X 0,Y 448.646,Z 702.53,A -85,B 0,C 180,E1 8148.774,E2 8148.774} C_VEL
LIN {X 0,Y 454.882,Z 715.976,A -85,B 0,C 180,E1 8149.677,E2 8149.677} C_VEL
LIN {X 0,Y 474.48,Z 756.104,A -85,B 0,C 180,E1 8152.215,E2 8152.215} C_VEL
LIN {X 0,Y 472.203,Z 796.625,A -85,B 0,C 180,E1 8153.357,E2 8153.357} C_VEL
LIN {X 0,Y 469.871,Z 825.231,A -85,B 0,C 180,E1 8154.637,E2 8154.637} C_VEL
LIN {X 0,Y 459.816,Z 854.749,A -85,B 0,C 180,E1 8155.953,E2 8155.953} C_VEL
LIN {X 0,Y 459.502,Z 856.6,A -85,B 0,C 180,E1 8156.078,E2 8156.078} C_VEL
LIN {X 0,Y 454.945,Z 892.496,A -85,B 0,C 180,E1 8159.121,E2 8159.121} C_VEL
LIN {X 0,Y 450.561,Z 924.731,A -85,B 0,C 180,E1 8162.808,E2 8162.808} C_VEL
LIN {X 0,Y 446.939,Z 953.118,A -85,B 0,C 180,E1 8167.152,E2 8167.152} C_VEL
LIN {X 0,Y 444.358,Z 975.365,A -85,B 0,C 180,E1 8171.693,E2 8171.693} C_VEL
LIN {X 0,Y 442.899,Z 991.036,A -85,B 0,C 180,E1 8176.202,E2 8176.202} C_VEL
LIN {X 0,Y 442.188,Z 1002.561,A -85,B 0,C 180,E1 8181.149,E2 8181.149} C_VEL
LIN {X 0,Y 441.92,Z 1008.907,A -85,B 0,C 180,E1 8186.084,E2 8186.084} C_VEL
LIN {X 0,Y 441.954,Z 1010.5,A -85,B 0,C 180,E1 8190,E2 8190} C_VEL
LIN {X 0,Y 441.91,Z 1008.91,A -85,B 0,C 180,E1 8193.916,E2 8193.916} C_VEL
LIN {X 0,Y 442.197,Z 1002.563,A -85,B 0,C 180,E1 8198.851,E2 8198.851} C_VEL
LIN {X 0,Y 442.987,Z 989.988,A -85,B 0,C 180,E1 8204.141,E2 8204.141} C_VEL
LIN {X 0,Y 444.454,Z 974.411,A -85,B 0,C 180,E1 8208.544,E2 8208.544} C_VEL
LIN {X 0,Y 447.233,Z 950.336,A -85,B 0,C 180,E1 8213.357,E2 8213.357} C_VEL
LIN {X 0,Y 450.859,Z 923.197,A -85,B 0,C 180,E1 8217.426,E2 8217.426} C_VEL
LIN {X 0,Y 455.229,Z 891.427,A -85,B 0,C 180,E1 8221.035,E2 8221.035} C_VEL
LIN {X 0,Y 459.817,Z 856.202,A -85,B 0,C 180,E1 8224.006,E2 8224.006} C_VEL
LIN {X 0,Y 463.827,Z 819.851,A -85,B 0,C 180,E1 8226.209,E2 8226.209} C_VEL
LIN {X 0,Y 466.996,Z 782.41,A -85,B 0,C 180,E1 8227.718,E2 8227.718} C_VEL
LIN {X 0,Y 467.861,Z 757.836,A -85,B 0,C 180,E1 8228.393,E2 8228.393} C_VEL
LIN {X 0,Y 442.914,Z 707.87,A -85,B 0,C 180,E1 8231.783,E2 8231.783} C_VEL
LIN {X 0,Y 440.84,Z 702.53,A -85,B 0,C 180,E1 8232.234,E2 8232.234} C_VEL
LIN {X 0,Y 440.655,Z 702.53,A -85,B 0,C 180,E1 8239.4,E2 8239.4} C_VEL
LIN {X 0,Y 440.797,Z 702.53,A -85,B 0,C 180,E1 8245.246,E2 8245.246} C_VEL
LIN {X 0,Y 440.939,Z 702.53,A -85,B 0,C 180,E1 8251.361,E2 8251.361} C_VEL
LIN {X 0,Y 441.018,Z 702.53,A -85,B 0,C 180,E1 8257.879,E2 8257.879} C_VEL
LIN {X 0,Y 441.298,Z 702.53,A -85,B 0,C 180,E1 8264.111,E2 8264.111} C_VEL
LIN {X 0,Y 441.491,Z 702.53,A -85,B 0,C 180,E1 8270.146,E2 8270.146} C_VEL
LIN {X 0,Y 441.752,Z 702.53,A -85,B 0,C 180,E1 8276.068,E2 8276.068} C_VEL
LIN {X 0,Y 441.908,Z 702.53,A -85,B 0,C 180,E1 8281.941,E2 8281.941} C_VEL
LIN {X 0,Y 441.574,Z 702.53,A -85,B 0,C 180,E1 8287.839,E2 8287.839} C_VEL
LIN {X 0,Y 441.36,Z 702.53,A -85,B 0,C 180,E1 8293.828,E2 8293.828} C_VEL
LIN {X 0,Y 441.123,Z 702.53,A -85,B 0,C 180,E1 8299.982,E2 8299.982} C_VEL
LIN {X 0,Y 440.906,Z 702.53,A -85,B 0,C 180,E1 8306.395,E2 8306.395} C_VEL
LIN {X 0,Y 440.744,Z 702.53,A -85,B 0,C 180,E1 8313.189,E2 8313.189} C_VEL
LIN {X 0,Y 440.81,Z 702.53,A -85,B 0,C 180,E1 8318.061,E2 8318.061} C_VEL
LIN {X 0,Y 440.682,Z 702.53,A -85,B 0,C 180,E1 8324.02,E2 8324.02} C_VEL
LIN {X 0,Y 440.633,Z 702.53,A -85,B 0,C 180,E1 8329.407,E2 8329.407} C_VEL
LIN {X 0,Y 440.797,Z 702.53,A -85,B 0,C 180,E1 8335.2,E2 8335.2} C_VEL
LIN {X 0,Y 440.922,Z 702.53,A -85,B 0,C 180,E1 8341.371,E2 8341.371} C_VEL
LIN {X 0,Y 441.083,Z 702.53,A -85,B 0,C 180,E1 8347.894,E2 8347.894} C_VEL
LIN {X 0,Y 441.289,Z 702.53,A -85,B 0,C 180,E1 8354.124,E2 8354.124} C_VEL
LIN {X 0,Y 441.489,Z 702.53,A -85,B 0,C 180,E1 8360.867,E2 8360.867} C_VEL
LIN {X 0,Y 447.645,Z 716.158,A -85,B 0,C 180,E1 8361.787,E2 8361.787} C_VEL
LIN {X 0,Y 460.868,Z 747.232,A -85,B 0,C 180,E1 8364.061,E2 8364.061} C_VEL
LIN {X 0,Y 462.076,Z 755.75,A -85,B 0,C 180,E1 8364.554,E2 8364.554} C_VEL
LIN {X 0,Y 458.886,Z 789.783,A -85,B 0,C 180,E1 8366.347,E2 8366.347} C_VEL
LIN {X 0,Y 455.06,Z 821.973,A -85,B 0,C 180,E1 8368.813,E2 8368.813} C_VEL
LIN {X 0,Y 451.173,Z 851.275,A -85,B 0,C 180,E1 8371.917,E2 8371.917} C_VEL
LIN {X 0,Y 447.481,Z 878.116,A -85,B 0,C 180,E1 8375.807,E2 8375.807} C_VEL
LIN {X 0,Y 444.776,Z 899.729,A -85,B 0,C 180,E1 8380.15,E2 8380.15} C_VEL
LIN {X 0,Y 443.082,Z 915.836,A -85,B 0,C 180,E1 8384.742,E2 8384.742} C_VEL
LIN {X 0,Y 442.398,Z 925.486,A -85,B 0,C 180,E1 8388.908,E2 8388.908} C_VEL
LIN {X 0,Y 441.846,Z 930.86,A -85,B 0,C 180,E1 8392.834,E2 8392.834} C_VEL
LIN {X 0,Y 441.498,Z 932.769,A -85,B 0,C 180,E1 8397.354,E2 8397.354} C_VEL
LIN {X 0,Y 441.931,Z 930.62,A -85,B 0,C 180,E1 8401.441,E2 8401.441} C_VEL
LIN {X 0,Y 442.568,Z 923.112,A -85,B 0,C 180,E1 8406.304,E2 8406.304} C_VEL
LIN {X 0,Y 443.596,Z 910.58,A -85,B 0,C 180,E1 8410.959,E2 8410.959} C_VEL
LIN {X 0,Y 445.673,Z 893.249,A -85,B 0,C 180,E1 8415.321,E2 8415.321} C_VEL
LIN {X 0,Y 448.863,Z 869.926,A -85,B 0,C 180,E1 8419.536,E2 8419.536} C_VEL
LIN {X 0,Y 452.722,Z 842.239,A -85,B 0,C 180,E1 8423.161,E2 8423.161} C_VEL
LIN {X 0,Y 456.91,Z 811.153,A -85,B 0,C 180,E1 8426.121,E2 8426.121} C_VEL
LIN {X 0,Y 460.726,Z 777.074,A -85,B 0,C 180,E1 8428.422,E2 8428.422} C_VEL
LIN {X 0,Y 462.31,Z 750.98,A -85,B 0,C 180,E1 8429.7,E2 8429.7} C_VEL
LIN {X 0,Y 448.052,Z 717.467,A -85,B 0,C 180,E1 8432.263,E2 8432.263} C_VEL
LIN {X 0,Y 441.084,Z 703.62,A -85,B 0,C 180,E1 8433.31,E2 8433.31} C_VEL
LIN {X 0,Y 441.009,Z 702.53,A -85,B 0,C 180,E1 8433.436,E2 8433.436} C_VEL
LIN {X 0,Y 441.197,Z 702.53,A -85,B 0,C 180,E1 8440.021,E2 8440.021} C_VEL
LIN {X 0,Y 441.446,Z 702.53,A -85,B 0,C 180,E1 8446.175,E2 8446.175} C_VEL
LIN {X 0,Y 441.536,Z 702.53,A -85,B 0,C 180,E1 8452.659,E2 8452.659} C_VEL
LIN {X 0,Y 441.708,Z 702.53,A -85,B 0,C 180,E1 8458.058,E2 8458.058} C_VEL
LIN {X 0,Y 441.677,Z 702.53,A -85,B 0,C 180,E1 8463.933,E2 8463.933} C_VEL
LIN {X 0,Y 441.417,Z 702.53,A -85,B 0,C 180,E1 8469.855,E2 8469.855} C_VEL
LIN {X 0,Y 441.195,Z 702.53,A -85,B 0,C 180,E1 8475.893,E2 8475.893} C_VEL
LIN {X 0,Y 440.982,Z 702.53,A -85,B 0,C 180,E1 8482.492,E2 8482.492} C_VEL
LIN {X 0,Y 440.822,Z 702.53,A -85,B 0,C 180,E1 8488.647,E2 8488.647} C_VEL
LIN {X 0,Y 440.78,Z 702.53,A -85,B 0,C 180,E1 8495.601,E2 8495.601} C_VEL
LIN {X 0,Y 440.712,Z 702.53,A -85,B 0,C 180,E1 8501.123,E2 8501.123} C_VEL
LIN {X 0,Y 440.71,Z 702.711,A -85,B 0,C 180,E1 8507.969,E2 8507.969} C_VEL
LIN {X 0,Y 445.585,Z 713.041,A -85,B 0,C 180,E1 8508.69,E2 8508.69} C_VEL
LIN {X 0,Y 467.898,Z 758.153,A -85,B 0,C 180,E1 8511.699,E2 8511.699} C_VEL
LIN {X 0,Y 465.345,Z 800.013,A -85,B 0,C 180,E1 8512.956,E2 8512.956} C_VEL
LIN {X 0,Y 461.471,Z 839.923,A -85,B 0,C 180,E1 8514.969,E2 8514.969} C_VEL
LIN {X 0,Y 459.502,Z 856.6,A -85,B 0,C 180,E1 8516.078,E2 8516.078} C_VEL
LIN {X 0,Y 454.078,Z 871.65,A -85,B 0,C 180,E1 8516.992,E2 8516.992} C_VEL
LIN {X 0,Y 448.649,Z 886.03,A -85,B 0,C 180,E1 8518.054,E2 8518.054} C_VEL
LIN {X 0,Y 444.062,Z 918.11,A -85,B 0,C 180,E1 8521.591,E2 8521.591} C_VEL
LIN {X 0,Y 440.138,Z 946.274,A -85,B 0,C 180,E1 8525.705,E2 8525.705} C_VEL
LIN {X 0,Y 437.153,Z 970.119,A -85,B 0,C 180,E1 8530.332,E2 8530.332} C_VEL
LIN {X 0,Y 435.348,Z 987.661,A -85,B 0,C 180,E1 8534.932,E2 8534.932} C_VEL
LIN {X 0,Y 434.506,Z 999.717,A -85,B 0,C 180,E1 8539.494,E2 8539.494} C_VEL
LIN {X 0,Y 434.086,Z 1006.953,A -85,B 0,C 180,E1 8544.013,E2 8544.013} C_VEL
LIN {X 0,Y 434.046,Z 1010.089,A -85,B 0,C 180,E1 8548.007,E2 8548.007} C_VEL
LIN {X 0,Y 434.087,Z 1010.09,A -85,B 0,C 180,E1 8551.992,E2 8551.992} C_VEL
LIN {X 0,Y 434.197,Z 1005.753,A -85,B 0,C 180,E1 8556.987,E2 8556.987} C_VEL
LIN {X 0,Y 434.764,Z 995.253,A -85,B 0,C 180,E1 8562.456,E2 8562.456} C_VEL
LIN {X 0,Y 436.243,Z 978.7,A -85,B 0,C 180,E1 8567.618,E2 8567.618} C_VEL
LIN {X 0,Y 438.744,Z 956.592,A -85,B 0,C 180,E1 8572.497,E2 8572.497} C_VEL
LIN {X 0,Y 442.413,Z 929.874,A -85,B 0,C 180,E1 8576.884,E2 8576.884} C_VEL
LIN {X 0,Y 446.831,Z 899.879,A -85,B 0,C 180,E1 8580.608,E2 8580.608} C_VEL
LIN {X 0,Y 451.521,Z 866.466,A -85,B 0,C 180,E1 8583.73,E2 8583.73} C_VEL
LIN {X 0,Y 455.965,Z 830.505,A -85,B 0,C 180,E1 8586.18,E2 8586.18} C_VEL
LIN {X 0,Y 459.747,Z 791.425,A -85,B 0,C 180,E1 8587.98,E2 8587.98} C_VEL
LIN {X 0,Y 461.247,Z 760.192,A -85,B 0,C 180,E1 8588.93,E2 8588.93} C_VEL
LIN {X 0,Y 437.787,Z 712.998,A -85,B 0,C 180,E1 8592.218,E2 8592.218} C_VEL
LIN {X 0,Y 432.923,Z 703.658,A -85,B 0,C 180,E1 8592.938,E2 8592.938} C_VEL
LIN {X 0,Y 432.844,Z 702.53,A -85,B 0,C 180,E1 8593.194,E2 8593.194} C_VEL
LIN {X 0,Y 432.687,Z 702.53,A -85,B 0,C 180,E1 8600.109,E2 8600.109} C_VEL
LIN {X 0,Y 432.892,Z 702.53,A -85,B 0,C 180,E1 8606.785,E2 8606.785} C_VEL
LIN {X 0,Y 433.013,Z 702.53,A -85,B 0,C 180,E1 8613.05,E2 8613.05} C_VEL
LIN {X 0,Y 433.215,Z 702.53,A -85,B 0,C 180,E1 8620.134,E2 8620.134} C_VEL
LIN {X 0,Y 433.437,Z 702.53,A -85,B 0,C 180,E1 8625.881,E2 8625.881} C_VEL
LIN {X 0,Y 433.633,Z 702.53,A -85,B 0,C 180,E1 8631.984,E2 8631.984} C_VEL
LIN {X 0,Y 433.826,Z 702.53,A -85,B 0,C 180,E1 8637.991,E2 8637.991} C_VEL
LIN {X 0,Y 433.773,Z 702.53,A -85,B 0,C 180,E1 8643.973,E2 8643.973} C_VEL
LIN {X 0,Y 433.53,Z 702.53,A -85,B 0,C 180,E1 8650.004,E2 8650.004} C_VEL
LIN {X 0,Y 433.328,Z 702.53,A -85,B 0,C 180,E1 8656.156,E2 8656.156} C_VEL
LIN {X 0,Y 433.143,Z 702.53,A -85,B 0,C 180,E1 8662.511,E2 8662.511} C_VEL
LIN {X 0,Y 432.866,Z 702.53,A -85,B 0,C 180,E1 8669.363,E2 8669.363} C_VEL
LIN {X 0,Y 432.819,Z 702.53,A -85,B 0,C 180,E1 8673.878,E2 8673.878} C_VEL
LIN {X 0,Y 432.802,Z 702.53,A -85,B 0,C 180,E1 8679.91,E2 8679.91} C_VEL
LIN {X 0,Y 432.758,Z 702.53,A -85,B 0,C 180,E1 8685.782,E2 8685.782} C_VEL
LIN {X 0,Y 432.72,Z 702.53,A -85,B 0,C 180,E1 8691.119,E2 8691.119} C_VEL
LIN {X 0,Y 432.919,Z 702.53,A -85,B 0,C 180,E1 8696.729,E2 8696.729} C_VEL
LIN {X 0,Y 433.03,Z 702.53,A -85,B 0,C 180,E1 8703.062,E2 8703.062} C_VEL
LIN {X 0,Y 433.274,Z 702.53,A -85,B 0,C 180,E1 8710.029,E2 8710.029} C_VEL
LIN {X 0,Y 433.42,Z 702.53,A -85,B 0,C 180,E1 8716.996,E2 8716.996} C_VEL
LIN {X 0,Y 433.565,Z 702.53,A -85,B 0,C 180,E1 8720.056,E2 8720.056} C_VEL
LIN {X 0,Y 440.279,Z 717.095,A -85,B 0,C 180,E1 8721.094,E2 8721.094} C_VEL
LIN {X 0,Y 453.804,Z 748.679,A -85,B 0,C 180,E1 8723.501,E2 8723.501} C_VEL
LIN {X 0,Y 455.459,Z 756.924,A -85,B 0,C 180,E1 8724.04,E2 8724.04} C_VEL
LIN {X 0,Y 451.967,Z 791.948,A -85,B 0,C 180,E1 8725.931,E2 8725.931} C_VEL
LIN {X 0,Y 447.842,Z 825.012,A -85,B 0,C 180,E1 8728.552,E2 8728.552} C_VEL
LIN {X 0,Y 443.477,Z 855.607,A -85,B 0,C 180,E1 8731.95,E2 8731.95} C_VEL
LIN {X 0,Y 439.663,Z 881.475,A -85,B 0,C 180,E1 8735.91,E2 8735.91} C_VEL
LIN {X 0,Y 436.922,Z 902.056,A -85,B 0,C 180,E1 8740.243,E2 8740.243} C_VEL
LIN {X 0,Y 435.156,Z 918.028,A -85,B 0,C 180,E1 8745.074,E2 8745.074} C_VEL
LIN {X 0,Y 434.529,Z 927.09,A -85,B 0,C 180,E1 8749.264,E2 8749.264} C_VEL
LIN {X 0,Y 434.026,Z 931.327,A -85,B 0,C 180,E1 8752.486,E2 8752.486} C_VEL
LIN {X 0,Y 433.628,Z 933.531,A -85,B 0,C 180,E1 8756.898,E2 8756.898} C_VEL
LIN {X 0,Y 434.143,Z 930.732,A -85,B 0,C 180,E1 8762.072,E2 8762.072} C_VEL
LIN {X 0,Y 434.728,Z 924.508,A -85,B 0,C 180,E1 8766.165,E2 8766.165} C_VEL
LIN {X 0,Y 435.877,Z 911.59,A -85,B 0,C 180,E1 8771.132,E2 8771.132} C_VEL
LIN {X 0,Y 438.021,Z 894.762,A -85,B 0,C 180,E1 8775.486,E2 8775.486} C_VEL
LIN {X 0,Y 441.244,Z 872.629,A -85,B 0,C 180,E1 8779.624,E2 8779.624} C_VEL
LIN {X 0,Y 445.401,Z 844.797,A -85,B 0,C 180,E1 8783.42,E2 8783.42} C_VEL
LIN {X 0,Y 449.728,Z 814.53,A -85,B 0,C 180,E1 8786.409,E2 8786.409} C_VEL
LIN {X 0,Y 453.579,Z 782.827,A -85,B 0,C 180,E1 8788.662,E2 8788.662} C_VEL
LIN {X 0,Y 455.735,Z 753.551,A -85,B 0,C 180,E1 8790.183,E2 8790.183} C_VEL
LIN {X 0,Y 441.521,Z 720.008,A -85,B 0,C 180,E1 8792.871,E2 8792.871} C_VEL
LIN {X 0,Y 433.191,Z 703.85,A -85,B 0,C 180,E1 8794.173,E2 8794.173} C_VEL
LIN {X 0,Y 433.09,Z 702.53,A -85,B 0,C 180,E1 8794.287,E2 8794.287} C_VEL
LIN {X 0,Y 433.309,Z 702.53,A -85,B 0,C 180,E1 8800.102,E2 8800.102} C_VEL
LIN {X 0,Y 433.535,Z 702.53,A -85,B 0,C 180,E1 8805.918,E2 8805.918} C_VEL
LIN {X 0,Y 433.589,Z 702.53,A -85,B 0,C 180,E1 8812.658,E2 8812.658} C_VEL
LIN {X 0,Y 433.804,Z 702.53,A -85,B 0,C 180,E1 8818.023,E2 8818.023} C_VEL
LIN {X 0,Y 433.771,Z 702.53,A -85,B 0,C 180,E1 8824.005,E2 8824.005} C_VEL
LIN {X 0,Y 433.488,Z 702.53,A -85,B 0,C 180,E1 8830.038,E2 8830.038} C_VEL
LIN {X 0,Y 433.277,Z 702.53,A -85,B 0,C 180,E1 8836.191,E2 8836.191} C_VEL
LIN {X 0,Y 433.089,Z 702.53,A -85,B 0,C 180,E1 8842.548,E2 8842.548} C_VEL
LIN {X 0,Y 432.82,Z 702.53,A -85,B 0,C 180,E1 8849.352,E2 8849.352} C_VEL
LIN {X 0,Y 432.812,Z 702.53,A -85,B 0,C 180,E1 8853.917,E2 8853.917} C_VEL
LIN {X 0,Y 432.762,Z 702.53,A -85,B 0,C 180,E1 8859.903,E2 8859.903} C_VEL
LIN {X 0,Y 432.729,Z 702.53,A -85,B 0,C 180,E1 8867.036,E2 8867.036} C_VEL
LIN {X 0,Y 437.672,Z 712.953,A -85,B 0,C 180,E1 8867.851,E2 8867.851} C_VEL
LIN {X 0,Y 461.171,Z 760.48,A -85,B 0,C 180,E1 8871.165,E2 8871.165} C_VEL
LIN {X 0,Y 458.507,Z 801.848,A -85,B 0,C 180,E1 8872.486,E2 8872.486} C_VEL
LIN {X 0,Y 454.535,Z 840.837,A -85,B 0,C 180,E1 8874.516,E2 8874.516} C_VEL
LIN {X 0,Y 449.968,Z 876.4,A -85,B 0,C 180,E1 8877.176,E2 8877.176} C_VEL
LIN {X 0,Y 448.649,Z 886.03,A -85,B 0,C 180,E1 8878.054,E2 8878.054} C_VEL
LIN {X 0,Y 443.066,Z 899.956,A -85,B 0,C 180,E1 8879.252,E2 8879.252} C_VEL
LIN {X 0,Y 437.402,Z 913.065,A -85,B 0,C 180,E1 8880.55,E2 8880.55} C_VEL
LIN {X 0,Y 432.869,Z 943.518,A -85,B 0,C 180,E1 8884.933,E2 8884.933} C_VEL
LIN {X 0,Y 429.555,Z 968.149,A -85,B 0,C 180,E1 8889.701,E2 8889.701} C_VEL
LIN {X 0,Y 427.516,Z 986.875,A -85,B 0,C 180,E1 8894.649,E2 8894.649} C_VEL
LIN {X 0,Y 426.565,Z 1000.322,A -85,B 0,C 180,E1 8899.812,E2 8899.812} C_VEL
LIN {X 0,Y 426.193,Z 1006.928,A -85,B 0,C 180,E1 8903.902,E2 8903.902} C_VEL
LIN {X 0,Y 426.141,Z 1010.088,A -85,B 0,C 180,E1 8907.97,E2 8907.97} C_VEL
LIN {X 0,Y 426.181,Z 1010.09,A -85,B 0,C 180,E1 8912.029,E2 8912.029} C_VEL
LIN {X 0,Y 426.286,Z 1004.952,A -85,B 0,C 180,E1 8917.593,E2 8917.593} C_VEL
LIN {X 0,Y 426.901,Z 994.734,A -85,B 0,C 180,E1 8922.643,E2 8922.643} C_VEL
LIN {X 0,Y 428.367,Z 979.262,A -85,B 0,C 180,E1 8927.612,E2 8927.612} C_VEL
LIN {X 0,Y 430.959,Z 957.194,A -85,B 0,C 180,E1 8932.654,E2 8932.654} C_VEL
LIN {X 0,Y 434.843,Z 930.584,A -85,B 0,C 180,E1 8937.155,E2 8937.155} C_VEL
LIN {X 0,Y 439.547,Z 900.459,A -85,B 0,C 180,E1 8940.995,E2 8940.995} C_VEL
LIN {X 0,Y 444.446,Z 867.494,A -85,B 0,C 180,E1 8944.154,E2 8944.154} C_VEL
LIN {X 0,Y 449.175,Z 831.276,A -85,B 0,C 180,E1 8946.681,E2 8946.681} C_VEL
LIN {X 0,Y 453.152,Z 792.744,A -85,B 0,C 180,E1 8948.503,E2 8948.503} C_VEL
LIN {X 0,Y 454.85,Z 763.056,A -85,B 0,C 180,E1 8949.433,E2 8949.433} C_VEL
LIN {X 0,Y 432.478,Z 717.728,A -85,B 0,C 180,E1 8952.69,E2 8952.69} C_VEL
LIN {X 0,Y 424.96,Z 703.388,A -85,B 0,C 180,E1 8953.837,E2 8953.837} C_VEL
LIN {X 0,Y 424.885,Z 702.53,A -85,B 0,C 180,E1 8953.928,E2 8953.928} C_VEL
LIN {X 0,Y 424.783,Z 702.53,A -85,B 0,C 180,E1 8960.24,E2 8960.24} C_VEL
LIN {X 0,Y 424.855,Z 702.53,A -85,B 0,C 180,E1 8965.358,E2 8965.358} C_VEL
LIN {X 0,Y 424.98,Z 702.53,A -85,B 0,C 180,E1 8970.18,E2 8970.18} C_VEL
LIN {X 0,Y 425.174,Z 702.53,A -85,B 0,C 180,E1 8977.337,E2 8977.337} C_VEL
LIN {X 0,Y 425.416,Z 702.53,A -85,B 0,C 180,E1 8983.501,E2 8983.501} C_VEL
LIN {X 0,Y 425.626,Z 702.53,A -85,B 0,C 180,E1 8989.775,E2 8989.775} C_VEL
LIN {X 0,Y 425.923,Z 702.53,A -85,B 0,C 180,E1 8995.921,E2 8995.921} C_VEL
LIN {X 0,Y 426.084,Z 702.53,A -85,B 0,C 180,E1 9002.013,E2 9002.013} C_VEL
LIN {X 0,Y 425.719,Z 702.53,A -85,B 0,C 180,E1 9008.133,E2 9008.133} C_VEL
LIN {X 0,Y 425.473,Z 702.53,A -85,B 0,C 180,E1 9014.355,E2 9014.355} C_VEL
LIN {X 0,Y 425.233,Z 702.53,A -85,B 0,C 180,E1 9020.763,E2 9020.763} C_VEL
LIN {X 0,Y 425.006,Z 702.53,A -85,B 0,C 180,E1 9027.463,E2 9027.463} C_VEL
LIN {X 0,Y 424.891,Z 702.53,A -85,B 0,C 180,E1 9032.162,E2 9032.162} C_VEL
LIN {X 0,Y 424.902,Z 702.53,A -85,B 0,C 180,E1 9038.619,E2 9038.619} C_VEL
LIN {X 0,Y 424.84,Z 702.53,A -85,B 0,C 180,E1 9045.23,E2 9045.23} C_VEL
LIN {X 0,Y 424.796,Z 702.53,A -85,B 0,C 180,E1 9051.357,E2 9051.357} C_VEL
LIN {X 0,Y 425.01,Z 702.53,A -85,B 0,C 180,E1 9058.391,E2 9058.391} C_VEL
LIN {X 0,Y 425.155,Z 702.53,A -85,B 0,C 180,E1 9064.791,E2 9064.791} C_VEL
LIN {X 0,Y 425.314,Z 702.53,A -85,B 0,C 180,E1 9071.378,E2 9071.378} C_VEL
LIN {X 0,Y 425.57,Z 702.53,A -85,B 0,C 180,E1 9077.717,E2 9077.717} C_VEL
LIN {X 0,Y 425.578,Z 702.53,A -85,B 0,C 180,E1 9079.208,E2 9079.208} C_VEL
LIN {X 0,Y 429.789,Z 712.03,A -85,B 0,C 180,E1 9079.889,E2 9079.889} C_VEL
LIN {X 0,Y 445.504,Z 746.111,A -85,B 0,C 180,E1 9082.619,E2 9082.619} C_VEL
LIN {X 0,Y 448.794,Z 758.742,A -85,B 0,C 180,E1 9083.537,E2 9083.537} C_VEL
LIN {X 0,Y 445.062,Z 794.106,A -85,B 0,C 180,E1 9085.503,E2 9085.503} C_VEL
LIN {X 0,Y 440.556,Z 828.045,A -85,B 0,C 180,E1 9088.283,E2 9088.283} C_VEL
LIN {X 0,Y 436.288,Z 856.351,A -85,B 0,C 180,E1 9091.519,E2 9091.519} C_VEL
LIN {X 0,Y 432.284,Z 881.822,A -85,B 0,C 180,E1 9095.471,E2 9095.471} C_VEL
LIN {X 0,Y 429.374,Z 902.434,A -85,B 0,C 180,E1 9099.865,E2 9099.865} C_VEL
LIN {X 0,Y 427.41,Z 918.653,A -85,B 0,C 180,E1 9104.831,E2 9104.831} C_VEL
LIN {X 0,Y 426.627,Z 928.492,A -85,B 0,C 180,E1 9109.598,E2 9109.598} C_VEL
LIN {X 0,Y 426.034,Z 932.534,A -85,B 0,C 180,E1 9113.012,E2 9113.012} C_VEL
LIN {X 0,Y 425.742,Z 934.144,A -85,B 0,C 180,E1 9117.672,E2 9117.672} C_VEL
LIN {X 0,Y 426.45,Z 930.382,A -85,B 0,C 180,E1 9123.119,E2 9123.119} C_VEL
LIN {X 0,Y 427.195,Z 921.985,A -85,B 0,C 180,E1 9127.87,E2 9127.87} C_VEL
LIN {X 0,Y 428.856,Z 907.58,A -85,B 0,C 180,E1 9132.808,E2 9132.808} C_VEL
LIN {X 0,Y 431.543,Z 888.781,A -85,B 0,C 180,E1 9137.251,E2 9137.251} C_VEL
LIN {X 0,Y 435.427,Z 864.315,A -85,B 0,C 180,E1 9141.436,E2 9141.436} C_VEL
LIN {X 0,Y 439.957,Z 835.413,A -85,B 0,C 180,E1 9145.017,E2 9145.017} C_VEL
LIN {X 0,Y 444.531,Z 803.107,A -85,B 0,C 180,E1 9147.905,E2 9147.905} C_VEL
LIN {X 0,Y 448.705,Z 767.506,A -85,B 0,C 180,E1 9150.101,E2 9150.101} C_VEL
LIN {X 0,Y 448.954,Z 755.651,A -85,B 0,C 180,E1 9150.726,E2 9150.726} C_VEL
LIN {X 0,Y 435.055,Z 722.465,A -85,B 0,C 180,E1 9153.5,E2 9153.5} C_VEL
LIN {X 0,Y 425.265,Z 703.436,A -85,B 0,C 180,E1 9155.103,E2 9155.103} C_VEL
LIN {X 0,Y 425.217,Z 702.53,A -85,B 0,C 180,E1 9155.38,E2 9155.38} C_VEL
LIN {X 0,Y 425.402,Z 702.53,A -85,B 0,C 180,E1 9161.404,E2 9161.404} C_VEL
LIN {X 0,Y 425.651,Z 702.53,A -85,B 0,C 180,E1 9167.738,E2 9167.738} C_VEL
LIN {X 0,Y 425.784,Z 702.53,A -85,B 0,C 180,E1 9173.914,E2 9173.914} C_VEL
LIN {X 0,Y 426.013,Z 702.53,A -85,B 0,C 180,E1 9180.016,E2 9180.016} C_VEL
LIN {X 0,Y 425.801,Z 702.53,A -85,B 0,C 180,E1 9186.118,E2 9186.118} C_VEL
LIN {X 0,Y 425.522,Z 702.53,A -85,B 0,C 180,E1 9192.299,E2 9192.299} C_VEL
LIN {X 0,Y 425.277,Z 702.53,A -85,B 0,C 180,E1 9198.636,E2 9198.636} C_VEL
LIN {X 0,Y 425.044,Z 702.53,A -85,B 0,C 180,E1 9205.228,E2 9205.228} C_VEL
LIN {X 0,Y 424.864,Z 702.53,A -85,B 0,C 180,E1 9212.203,E2 9212.203} C_VEL
LIN {X 0,Y 424.87,Z 702.53,A -85,B 0,C 180,E1 9218.612,E2 9218.612} C_VEL
LIN {X 0,Y 424.775,Z 702.53,A -85,B 0,C 180,E1 9225.286,E2 9225.286} C_VEL
LIN {X 0,Y 424.824,Z 703.143,A -85,B 0,C 180,E1 9226.171,E2 9226.171} C_VEL
LIN {X 0,Y 449.217,Z 751.287,A -85,B 0,C 180,E1 9229.832,E2 9229.832} C_VEL
LIN {X 0,Y 454.809,Z 763.508,A -85,B 0,C 180,E1 9230.676,E2 9230.676} C_VEL
LIN {X 0,Y 451.774,Z 803.468,A -85,B 0,C 180,E1 9231.995,E2 9231.995} C_VEL
LIN {X 0,Y 447.734,Z 840.916,A -85,B 0,C 180,E1 9233.995,E2 9233.995} C_VEL
LIN {X 0,Y 442.887,Z 876.569,A -85,B 0,C 180,E1 9236.71,E2 9236.71} C_VEL
LIN {X 0,Y 437.919,Z 909.701,A -85,B 0,C 180,E1 9240.149,E2 9240.149} C_VEL
LIN {X 0,Y 437.402,Z 913.065,A -85,B 0,C 180,E1 9240.55,E2 9240.55} C_VEL
LIN {X 0,Y 431.75,Z 925.559,A -85,B 0,C 180,E1 9241.994,E2 9241.994} C_VEL
LIN {X 0,Y 426.182,Z 937.232,A -85,B 0,C 180,E1 9243.578,E2 9243.578} C_VEL
LIN {X 0,Y 422.432,Z 962.545,A -85,B 0,C 180,E1 9248.256,E2 9248.256} C_VEL
LIN {X 0,Y 420.139,Z 981.379,A -85,B 0,C 180,E1 9252.926,E2 9252.926} C_VEL
LIN {X 0,Y 418.87,Z 996.14,A -85,B 0,C 180,E1 9258.044,E2 9258.044} C_VEL
LIN {X 0,Y 418.384,Z 1004.633,A -85,B 0,C 180,E1 9262.528,E2 9262.528} C_VEL
LIN {X 0,Y 418.255,Z 1009.578,A -85,B 0,C 180,E1 9267.932,E2 9267.932} C_VEL
LIN {X 0,Y 418.292,Z 1009.587,A -85,B 0,C 180,E1 9272.067,E2 9272.067} C_VEL
LIN {X 0,Y 418.384,Z 1004.668,A -85,B 0,C 180,E1 9277.469,E2 9277.469} C_VEL
LIN {X 0,Y 418.972,Z 995.004,A -85,B 0,C 180,E1 9282.48,E2 9282.48} C_VEL
LIN {X 0,Y 420.545,Z 978.88,A -85,B 0,C 180,E1 9287.849,E2 9287.849} C_VEL
LIN {X 0,Y 423.433,Z 956.426,A -85,B 0,C 180,E1 9293.08,E2 9293.08} C_VEL
LIN {X 0,Y 427.442,Z 930.446,A -85,B 0,C 180,E1 9297.559,E2 9297.559} C_VEL
LIN {X 0,Y 432.48,Z 899.58,A -85,B 0,C 180,E1 9301.559,E2 9301.559} C_VEL
LIN {X 0,Y 437.656,Z 866.862,A -85,B 0,C 180,E1 9304.724,E2 9304.724} C_VEL
LIN {X 0,Y 442.626,Z 830.652,A -85,B 0,C 180,E1 9307.276,E2 9307.276} C_VEL
LIN {X 0,Y 446.745,Z 792.462,A -85,B 0,C 180,E1 9309.1,E2 9309.1} C_VEL
LIN {X 0,Y 448.405,Z 765.969,A -85,B 0,C 180,E1 9309.955,E2 9309.955} C_VEL
LIN {X 0,Y 427.916,Z 723.536,A -85,B 0,C 180,E1 9313.069,E2 9313.069} C_VEL
LIN {X 0,Y 416.985,Z 703.459,A -85,B 0,C 180,E1 9314.774,E2 9314.774} C_VEL
LIN {X 0,Y 416.941,Z 702.53,A -85,B 0,C 180,E1 9315.056,E2 9315.056} C_VEL
LIN {X 0,Y 416.851,Z 702.53,A -85,B 0,C 180,E1 9322.008,E2 9322.008} C_VEL
LIN {X 0,Y 416.945,Z 702.53,A -85,B 0,C 180,E1 9327.109,E2 9327.109} C_VEL
LIN {X 0,Y 417.061,Z 702.53,A -85,B 0,C 180,E1 9331.93,E2 9331.93} C_VEL
LIN {X 0,Y 417.288,Z 702.53,A -85,B 0,C 180,E1 9338.787,E2 9338.787} C_VEL
LIN {X 0,Y 417.571,Z 702.53,A -85,B 0,C 180,E1 9345.333,E2 9345.333} C_VEL
LIN {X 0,Y 417.782,Z 702.53,A -85,B 0,C 180,E1 9351.678,E2 9351.678} C_VEL
LIN {X 0,Y 418.047,Z 702.53,A -85,B 0,C 180,E1 9357.915,E2 9357.915} C_VEL
LIN {X 0,Y 417.952,Z 702.53,A -85,B 0,C 180,E1 9364.123,E2 9364.123} C_VEL
LIN {X 0,Y 417.675,Z 702.53,A -85,B 0,C 180,E1 9370.388,E2 9370.388} C_VEL
LIN {X 0,Y 417.448,Z 702.53,A -85,B 0,C 180,E1 9376.788,E2 9376.788} C_VEL
LIN {X 0,Y 417.202,Z 702.53,A -85,B 0,C 180,E1 9383.421,E2 9383.421} C_VEL
LIN {X 0,Y 416.988,Z 702.53,A -85,B 0,C 180,E1 9390.413,E2 9390.413} C_VEL
LIN {X 0,Y 416.978,Z 702.53,A -85,B 0,C 180,E1 9397.936,E2 9397.936} C_VEL
LIN {X 0,Y 416.877,Z 702.53,A -85,B 0,C 180,E1 9403.617,E2 9403.617} C_VEL
LIN {X 0,Y 416.822,Z 702.53,A -85,B 0,C 180,E1 9409.446,E2 9409.446} C_VEL
LIN {X 0,Y 416.931,Z 702.53,A -85,B 0,C 180,E1 9414.613,E2 9414.613} C_VEL
LIN {X 0,Y 417.109,Z 702.53,A -85,B 0,C 180,E1 9421.945,E2 9421.945} C_VEL
LIN {X 0,Y 417.311,Z 702.53,A -85,B 0,C 180,E1 9428.801,E2 9428.801} C_VEL
LIN {X 0,Y 417.566,Z 702.53,A -85,B 0,C 180,E1 9435.347,E2 9435.347} C_VEL
LIN {X 0,Y 417.668,Z 702.641,A -85,B 0,C 180,E1 9438.34,E2 9438.34} C_VEL
LIN {X 0,Y 422.229,Z 712.62,A -85,B 0,C 180,E1 9439.088,E2 9439.088} C_VEL
LIN {X 0,Y 438.071,Z 746.591,A -85,B 0,C 180,E1 9441.926,E2 9441.926} C_VEL
LIN {X 0,Y 442.137,Z 761.27,A -85,B 0,C 180,E1 9443.055,E2 9443.055} C_VEL
LIN {X 0,Y 438.213,Z 796.218,A -85,B 0,C 180,E1 9445.061,E2 9445.061} C_VEL
LIN {X 0,Y 433.472,Z 829.687,A -85,B 0,C 180,E1 9447.881,E2 9447.881} C_VEL
LIN {X 0,Y 428.883,Z 858.583,A -85,B 0,C 180,E1 9451.281,E2 9451.281} C_VEL
LIN {X 0,Y 424.629,Z 884.058,A -85,B 0,C 180,E1 9455.364,E2 9455.364} C_VEL
LIN {X 0,Y 421.446,Z 905.019,A -85,B 0,C 180,E1 9460.041,E2 9460.041} C_VEL
LIN {X 0,Y 419.659,Z 919.278,A -85,B 0,C 180,E1 9464.579,E2 9464.579} C_VEL
LIN {X 0,Y 418.881,Z 928.385,A -85,B 0,C 180,E1 9468.919,E2 9468.919} C_VEL
LIN {X 0,Y 418.117,Z 933.602,A -85,B 0,C 180,E1 9473.391,E2 9473.391} C_VEL
LIN {X 0,Y 417.882,Z 934.809,A -85,B 0,C 180,E1 9477.999,E2 9477.999} C_VEL
LIN {X 0,Y 418.526,Z 931.648,A -85,B 0,C 180,E1 9482.741,E2 9482.741} C_VEL
LIN {X 0,Y 419.347,Z 923.479,A -85,B 0,C 180,E1 9487.716,E2 9487.716} C_VEL
LIN {X 0,Y 421.116,Z 909.028,A -85,B 0,C 180,E1 9492.91,E2 9492.91} C_VEL
LIN {X 0,Y 423.992,Z 890.245,A -85,B 0,C 180,E1 9497.485,E2 9497.485} C_VEL
LIN {X 0,Y 428.013,Z 866.386,A -85,B 0,C 180,E1 9501.684,E2 9501.684} C_VEL
LIN {X 0,Y 432.855,Z 837.428,A -85,B 0,C 180,E1 9505.393,E2 9505.393} C_VEL
LIN {X 0,Y 437.652,Z 805.552,A -85,B 0,C 180,E1 9508.324,E2 9508.324} C_VEL
LIN {X 0,Y 441.988,Z 770.379,A -85,B 0,C 180,E1 9510.57,E2 9510.57} C_VEL
LIN {X 0,Y 442.359,Z 758.153,A -85,B 0,C 180,E1 9511.241,E2 9511.241} C_VEL
LIN {X 0,Y 428.931,Z 725.775,A -85,B 0,C 180,E1 9514.076,E2 9514.076} C_VEL
LIN {X 0,Y 417.306,Z 703.133,A -85,B 0,C 180,E1 9516.09,E2 9516.09} C_VEL
LIN {X 0,Y 417.44,Z 702.53,A -85,B 0,C 180,E1 9521.036,E2 9521.036} C_VEL
LIN {X 0,Y 417.716,Z 702.53,A -85,B 0,C 180,E1 9527.502,E2 9527.502} C_VEL
LIN {X 0,Y 417.868,Z 702.53,A -85,B 0,C 180,E1 9533.799,E2 9533.799} C_VEL
LIN {X 0,Y 418.122,Z 702.53,A -85,B 0,C 180,E1 9540.017,E2 9540.017} C_VEL
LIN {X 0,Y 417.885,Z 702.53,A -85,B 0,C 180,E1 9546.234,E2 9546.234} C_VEL
LIN {X 0,Y 417.567,Z 702.53,A -85,B 0,C 180,E1 9552.645,E2 9552.645} C_VEL
LIN {X 0,Y 417.321,Z 702.53,A -85,B 0,C 180,E1 9559.005,E2 9559.005} C_VEL
LIN {X 0,Y 417.081,Z 702.53,A -85,B 0,C 180,E1 9565.744,E2 9565.744} C_VEL
LIN {X 0,Y 416.932,Z 702.53,A -85,B 0,C 180,E1 9570.456,E2 9570.456} C_VEL
LIN {X 0,Y 416.974,Z 702.53,A -85,B 0,C 180,E1 9577.979,E2 9577.979} C_VEL
LIN {X 0,Y 416.874,Z 702.53,A -85,B 0,C 180,E1 9585.161,E2 9585.161} C_VEL
LIN {X 0,Y 419.332,Z 708.259,A -85,B 0,C 180,E1 9585.61,E2 9585.61} C_VEL
LIN {X 0,Y 440.574,Z 748.818,A -85,B 0,C 180,E1 9588.905,E2 9588.905} C_VEL
LIN {X 0,Y 448.279,Z 767.813,A -85,B 0,C 180,E1 9590.191,E2 9590.191} C_VEL
LIN {X 0,Y 444.908,Z 806.833,A -85,B 0,C 180,E1 9591.563,E2 9591.563} C_VEL
LIN {X 0,Y 440.219,Z 846.842,A -85,B 0,C 180,E1 9593.839,E2 9593.839} C_VEL
LIN {X 0,Y 434.792,Z 883.547,A -85,B 0,C 180,E1 9596.863,E2 9596.863} C_VEL
LIN {X 0,Y 429.557,Z 916.195,A -85,B 0,C 180,E1 9600.54,E2 9600.54} C_VEL
LIN {X 0,Y 426.182,Z 937.232,A -85,B 0,C 180,E1 9603.578,E2 9603.578} C_VEL
LIN {X 0,Y 420.786,Z 948.206,A -85,B 0,C 180,E1 9605.28,E2 9605.28} C_VEL
LIN {X 0,Y 415.311,Z 958.308,A -85,B 0,C 180,E1 9607.106,E2 9607.106} C_VEL
LIN {X 0,Y 412.608,Z 978.508,A -85,B 0,C 180,E1 9611.983,E2 9611.983} C_VEL
LIN {X 0,Y 411.092,Z 994.164,A -85,B 0,C 180,E1 9617.276,E2 9617.276} C_VEL
LIN {X 0,Y 410.516,Z 1004.054,A -85,B 0,C 180,E1 9622.483,E2 9622.483} C_VEL
LIN {X 0,Y 410.378,Z 1008.867,A -85,B 0,C 180,E1 9627.892,E2 9627.892} C_VEL
LIN {X 0,Y 410.413,Z 1008.883,A -85,B 0,C 180,E1 9632.107,E2 9632.107} C_VEL
LIN {X 0,Y 410.521,Z 1004.09,A -85,B 0,C 180,E1 9637.531,E2 9637.531} C_VEL
LIN {X 0,Y 411.142,Z 994.291,A -85,B 0,C 180,E1 9642.722,E2 9642.722} C_VEL
LIN {X 0,Y 412.718,Z 978.591,A -85,B 0,C 180,E1 9648.065,E2 9648.065} C_VEL
LIN {X 0,Y 415.612,Z 957.323,A -85,B 0,C 180,E1 9653.194,E2 9653.194} C_VEL
LIN {X 0,Y 420.098,Z 929.896,A -85,B 0,C 180,E1 9658.04,E2 9658.04} C_VEL
LIN {X 0,Y 425.273,Z 899.778,A -85,B 0,C 180,E1 9662.018,E2 9662.018} C_VEL
LIN {X 0,Y 430.847,Z 866.373,A -85,B 0,C 180,E1 9665.303,E2 9665.303} C_VEL
LIN {X 0,Y 436.058,Z 830.407,A -85,B 0,C 180,E1 9667.867,E2 9667.867} C_VEL
LIN {X 0,Y 440.434,Z 791.461,A -85,B 0,C 180,E1 9669.737,E2 9669.737} C_VEL
LIN {X 0,Y 441.811,Z 768.417,A -85,B 0,C 180,E1 9670.52,E2 9670.52} C_VEL
LIN {X 0,Y 423.828,Z 730.599,A -85,B 0,C 180,E1 9673.376,E2 9673.376} C_VEL
LIN {X 0,Y 409.011,Z 703.156,A -85,B 0,C 180,E1 9675.762,E2 9675.762} C_VEL
LIN {X 0,Y 408.854,Z 702.53,A -85,B 0,C 180,E1 9681.127,E2 9681.127} C_VEL
LIN {X 0,Y 409.031,Z 702.53,A -85,B 0,C 180,E1 9686.389,E2 9686.389} C_VEL
LIN {X 0,Y 409.151,Z 702.53,A -85,B 0,C 180,E1 9693.719,E2 9693.719} C_VEL
LIN {X 0,Y 409.422,Z 702.53,A -85,B 0,C 180,E1 9700.614,E2 9700.614} C_VEL
LIN {X 0,Y 409.742,Z 702.53,A -85,B 0,C 180,E1 9707.22,E2 9707.22} C_VEL
LIN {X 0,Y 409.977,Z 702.53,A -85,B 0,C 180,E1 9713.645,E2 9713.645} C_VEL
LIN {X 0,Y 410.217,Z 702.53,A -85,B 0,C 180,E1 9719.983,E2 9719.983} C_VEL
LIN {X 0,Y 410.012,Z 702.53,A -85,B 0,C 180,E1 9726.428,E2 9726.428} C_VEL
LIN {X 0,Y 409.724,Z 702.53,A -85,B 0,C 180,E1 9732.746,E2 9732.746} C_VEL
LIN {X 0,Y 409.425,Z 702.53,A -85,B 0,C 180,E1 9739.35,E2 9739.35} C_VEL
LIN {X 0,Y 409.146,Z 702.53,A -85,B 0,C 180,E1 9746.243,E2 9746.243} C_VEL
LIN {X 0,Y 408.991,Z 702.53,A -85,B 0,C 180,E1 9753.574,E2 9753.574} C_VEL
LIN {X 0,Y 408.949,Z 702.53,A -85,B 0,C 180,E1 9759.204,E2 9759.204} C_VEL
LIN {X 0,Y 408.852,Z 702.53,A -85,B 0,C 180,E1 9765.472,E2 9765.472} C_VEL
LIN {X 0,Y 408.875,Z 702.53,A -85,B 0,C 180,E1 9771.141,E2 9771.141} C_VEL
LIN {X 0,Y 409.025,Z 702.53,A -85,B 0,C 180,E1 9778,E2 9778} C_VEL
LIN {X 0,Y 409.201,Z 702.53,A -85,B 0,C 180,E1 9783.735,E2 9783.735} C_VEL
LIN {X 0,Y 409.429,Z 702.53,A -85,B 0,C 180,E1 9790.628,E2 9790.628} C_VEL
LIN {X 0,Y 409.742,Z 702.53,A -85,B 0,C 180,E1 9797.375,E2 9797.375} C_VEL
LIN {X 0,Y 414.679,Z 713.061,A -85,B 0,C 180,E1 9798.245,E2 9798.245} C_VEL
LIN {X 0,Y 430.648,Z 747.037,A -85,B 0,C 180,E1 9801.203,E2 9801.203} C_VEL
LIN {X 0,Y 435.576,Z 762.931,A -85,B 0,C 180,E1 9802.519,E2 9802.519} C_VEL
LIN {X 0,Y 431.388,Z 798.337,A -85,B 0,C 180,E1 9804.606,E2 9804.606} C_VEL
LIN {X 0,Y 426.424,Z 831.319,A -85,B 0,C 180,E1 9807.465,E2 9807.465} C_VEL
LIN {X 0,Y 421.688,Z 859.485,A -85,B 0,C 180,E1 9810.846,E2 9810.846} C_VEL
LIN {X 0,Y 417.386,Z 883.865,A -85,B 0,C 180,E1 9814.802,E2 9814.802} C_VEL
LIN {X 0,Y 413.976,Z 905.113,A -85,B 0,C 180,E1 9819.559,E2 9819.559} C_VEL
LIN {X 0,Y 411.967,Z 919.528,A -85,B 0,C 180,E1 9824.165,E2 9824.165} C_VEL
LIN {X 0,Y 410.983,Z 929.849,A -85,B 0,C 180,E1 9829.297,E2 9829.297} C_VEL
LIN {X 0,Y 410.183,Z 934.679,A -85,B 0,C 180,E1 9833.871,E2 9833.871} C_VEL
LIN {X 0,Y 410.03,Z 935.439,A -85,B 0,C 180,E1 9838.584,E2 9838.584} C_VEL
LIN {X 0,Y 410.785,Z 931.741,A -85,B 0,C 180,E1 9843.438,E2 9843.438} C_VEL
LIN {X 0,Y 411.72,Z 922.872,A -85,B 0,C 180,E1 9848.542,E2 9848.542} C_VEL
LIN {X 0,Y 413.607,Z 908.969,A -85,B 0,C 180,E1 9853.45,E2 9853.45} C_VEL
LIN {X 0,Y 416.804,Z 889.599,A -85,B 0,C 180,E1 9858.171,E2 9858.171} C_VEL
LIN {X 0,Y 421.29,Z 864.739,A -85,B 0,C 180,E1 9862.519,E2 9862.519} C_VEL
LIN {X 0,Y 426.417,Z 835.475,A -85,B 0,C 180,E1 9866.204,E2 9866.204} C_VEL
LIN {X 0,Y 431.488,Z 803.179,A -85,B 0,C 180,E1 9869.131,E2 9869.131} C_VEL
LIN {X 0,Y 436.095,Z 766.578,A -85,B 0,C 180,E1 9871.403,E2 9871.403} C_VEL
LIN {X 0,Y 435.493,Z 759.808,A -85,B 0,C 180,E1 9871.853,E2 9871.853} C_VEL
LIN {X 0,Y 422.337,Z 727.767,A -85,B 0,C 180,E1 9874.777,E2 9874.777} C_VEL
LIN {X 0,Y 409.425,Z 703.409,A -85,B 0,C 180,E1 9877.119,E2 9877.119} C_VEL
LIN {X 0,Y 409.388,Z 702.53,A -85,B 0,C 180,E1 9877.149,E2 9877.149} C_VEL
LIN {X 0,Y 409.661,Z 702.53,A -85,B 0,C 180,E1 9883.284,E2 9883.284} C_VEL
LIN {X 0,Y 409.836,Z 702.53,A -85,B 0,C 180,E1 9889.411,E2 9889.411} C_VEL
LIN {X 0,Y 410.057,Z 702.53,A -85,B 0,C 180,E1 9895.797,E2 9895.797} C_VEL
LIN {X 0,Y 410.286,Z 702.53,A -85,B 0,C 180,E1 9902.124,E2 9902.124} C_VEL
LIN {X 0,Y 409.819,Z 702.53,A -85,B 0,C 180,E1 9908.485,E2 9908.485} C_VEL
LIN {X 0,Y 409.535,Z 702.53,A -85,B 0,C 180,E1 9914.961,E2 9914.961} C_VEL
LIN {X 0,Y 409.305,Z 702.53,A -85,B 0,C 180,E1 9921.647,E2 9921.647} C_VEL
LIN {X 0,Y 409.052,Z 702.53,A -85,B 0,C 180,E1 9928.67,E2 9928.67} C_VEL
LIN {X 0,Y 409.02,Z 702.53,A -85,B 0,C 180,E1 9936.189,E2 9936.189} C_VEL
LIN {X 0,Y 408.933,Z 702.53,A -85,B 0,C 180,E1 9943.423,E2 9943.423} C_VEL
LIN {X 0,Y 408.934,Z 702.53,A -85,B 0,C 180,E1 9944.111,E2 9944.111} C_VEL
LIN {X 0,Y 411.44,Z 708.232,A -85,B 0,C 180,E1 9944.592,E2 9944.592} C_VEL
LIN {X 0,Y 431.433,Z 745.325,A -85,B 0,C 180,E1 9947.844,E2 9947.844} C_VEL
LIN {X 0,Y 441.871,Z 769.943,A -85,B 0,C 180,E1 9949.63,E2 9949.63} C_VEL
LIN {X 0,Y 437.99,Z 811.007,A -85,B 0,C 180,E1 9951.166,E2 9951.166} C_VEL
LIN {X 0,Y 432.985,Z 849.853,A -85,B 0,C 180,E1 9953.502,E2 9953.502} C_VEL
LIN {X 0,Y 427.46,Z 885.332,A -85,B 0,C 180,E1 9956.546,E2 9956.546} C_VEL
LIN {X 0,Y 421.959,Z 917.666,A -85,B 0,C 180,E1 9960.313,E2 9960.313} C_VEL
LIN {X 0,Y 417.281,Z 945.888,A -85,B 0,C 180,E1 9964.71,E2 9964.71} C_VEL
LIN {X 0,Y 415.311,Z 958.308,A -85,B 0,C 180,E1 9967.106,E2 9967.106} C_VEL
LIN {X 0,Y 410.074,Z 967.537,A -85,B 0,C 180,E1 9969.058,E2 9969.058} C_VEL
LIN {X 0,Y 405.097,Z 975.872,A -85,B 0,C 180,E1 9971.112,E2 9971.112} C_VEL
LIN {X 0,Y 403.351,Z 992.386,A -85,B 0,C 180,E1 9976.603,E2 9976.603} C_VEL
LIN {X 0,Y 402.65,Z 1003.029,A -85,B 0,C 180,E1 9982.144,E2 9982.144} C_VEL
LIN {X 0,Y 402.531,Z 1008.159,A -85,B 0,C 180,E1 9987.851,E2 9987.851} C_VEL
LIN {X 0,Y 402.563,Z 1008.184,A -85,B 0,C 180,E1 9992.148,E2 9992.148} C_VEL
LIN {X 0,Y 402.65,Z 1003.119,A -85,B 0,C 180,E1 9997.854,E2 9997.854} C_VEL
LIN {X 0,Y 403.413,Z 992.467,A -85,B 0,C 180,E1 10003.435,E2 10003.435} C_VEL
LIN {X 0,Y 405.146,Z 975.793,A -85,B 0,C 180,E1 10008.999,E2 10008.999} C_VEL
LIN {X 0,Y 408.462,Z 953.846,A -85,B 0,C 180,E1 10014.194,E2 10014.194} C_VEL
LIN {X 0,Y 412.997,Z 928.15,A -85,B 0,C 180,E1 10018.717,E2 10018.717} C_VEL
LIN {X 0,Y 418.524,Z 897.777,A -85,B 0,C 180,E1 10022.74,E2 10022.74} C_VEL
LIN {X 0,Y 424.184,Z 865.343,A -85,B 0,C 180,E1 10025.943,E2 10025.943} C_VEL
LIN {X 0,Y 429.61,Z 829.665,A -85,B 0,C 180,E1 10028.499,E2 10028.499} C_VEL
LIN {X 0,Y 434.076,Z 791.34,A -85,B 0,C 180,E1 10030.361,E2 10030.361} C_VEL
LIN {X 0,Y 435.522,Z 771.357,A -85,B 0,C 180,E1 10031.058,E2 10031.058} C_VEL
LIN {X 0,Y 417.659,Z 733.285,A -85,B 0,C 180,E1 10034.031,E2 10034.031} C_VEL
LIN {X 0,Y 401.122,Z 703.782,A -85,B 0,C 180,E1 10036.767,E2 10036.767} C_VEL
LIN {X 0,Y 401.001,Z 702.53,A -85,B 0,C 180,E1 10036.952,E2 10036.952} C_VEL
LIN {X 0,Y 400.941,Z 702.53,A -85,B 0,C 180,E1 10042.961,E2 10042.961} C_VEL
LIN {X 0,Y 401.115,Z 702.53,A -85,B 0,C 180,E1 10049.914,E2 10049.914} C_VEL
LIN {X 0,Y 401.258,Z 702.53,A -85,B 0,C 180,E1 10055.551,E2 10055.551} C_VEL
LIN {X 0,Y 401.587,Z 702.53,A -85,B 0,C 180,E1 10062.492,E2 10062.492} C_VEL
LIN {X 0,Y 401.858,Z 702.53,A -85,B 0,C 180,E1 10069.163,E2 10069.163} C_VEL
LIN {X 0,Y 402.193,Z 702.53,A -85,B 0,C 180,E1 10075.68,E2 10075.68} C_VEL
LIN {X 0,Y 402.394,Z 702.53,A -85,B 0,C 180,E1 10082.131,E2 10082.131} C_VEL
LIN {X 0,Y 401.957,Z 702.53,A -85,B 0,C 180,E1 10088.617,E2 10088.617} C_VEL
LIN {X 0,Y 401.68,Z 702.53,A -85,B 0,C 180,E1 10095.225,E2 10095.225} C_VEL
LIN {X 0,Y 401.394,Z 702.53,A -85,B 0,C 180,E1 10102.059,E2 10102.059} C_VEL
LIN {X 0,Y 401.098,Z 702.53,A -85,B 0,C 180,E1 10109.253,E2 10109.253} C_VEL
LIN {X 0,Y 401.068,Z 702.53,A -85,B 0,C 180,E1 10114.329,E2 10114.329} C_VEL
LIN {X 0,Y 400.961,Z 702.53,A -85,B 0,C 180,E1 10121.175,E2 10121.175} C_VEL
LIN {X 0,Y 400.912,Z 702.53,A -85,B 0,C 180,E1 10127.351,E2 10127.351} C_VEL
LIN {X 0,Y 400.96,Z 702.53,A -85,B 0,C 180,E1 10132.975,E2 10132.975} C_VEL
LIN {X 0,Y 401.122,Z 702.53,A -85,B 0,C 180,E1 10139.855,E2 10139.855} C_VEL
LIN {X 0,Y 401.348,Z 702.53,A -85,B 0,C 180,E1 10145.57,E2 10145.57} C_VEL
LIN {X 0,Y 401.558,Z 702.53,A -85,B 0,C 180,E1 10152.505,E2 10152.505} C_VEL
LIN {X 0,Y 401.745,Z 702.989,A -85,B 0,C 180,E1 10156.435,E2 10156.435} C_VEL
LIN {X 0,Y 409.456,Z 718.038,A -85,B 0,C 180,E1 10157.77,E2 10157.77} C_VEL
LIN {X 0,Y 424.453,Z 750.688,A -85,B 0,C 180,E1 10160.739,E2 10160.739} C_VEL
LIN {X 0,Y 428.902,Z 765.904,A -85,B 0,C 180,E1 10162.027,E2 10162.027} C_VEL
LIN {X 0,Y 424.398,Z 801.314,A -85,B 0,C 180,E1 10164.211,E2 10164.211} C_VEL
LIN {X 0,Y 419.182,Z 834.148,A -85,B 0,C 180,E1 10167.163,E2 10167.163} C_VEL
LIN {X 0,Y 413.921,Z 863.666,A -85,B 0,C 180,E1 10170.863,E2 10170.863} C_VEL
LIN {X 0,Y 409.316,Z 888.409,A -85,B 0,C 180,E1 10175.147,E2 10175.147} C_VEL
LIN {X 0,Y 406.085,Z 907.412,A -85,B 0,C 180,E1 10179.689,E2 10179.689} C_VEL
LIN {X 0,Y 404.052,Z 921.614,A -85,B 0,C 180,E1 10184.505,E2 10184.505} C_VEL
LIN {X 0,Y 403.06,Z 931.307,A -85,B 0,C 180,E1 10189.692,E2 10189.692} C_VEL
LIN {X 0,Y 402.232,Z 935.653,A -85,B 0,C 180,E1 10194.374,E2 10194.374} C_VEL
LIN {X 0,Y 402.197,Z 935.904,A -85,B 0,C 180,E1 10199.193,E2 10199.193} C_VEL
LIN {X 0,Y 403.071,Z 931.661,A -85,B 0,C 180,E1 10204.165,E2 10204.165} C_VEL
LIN {X 0,Y 404.158,Z 922.139,A -85,B 0,C 180,E1 10209.401,E2 10209.401} C_VEL
LIN {X 0,Y 406.375,Z 907.497,A -85,B 0,C 180,E1 10214.424,E2 10214.424} C_VEL
LIN {X 0,Y 410.089,Z 886.495,A -85,B 0,C 180,E1 10219.379,E2 10219.379} C_VEL
LIN {X 0,Y 415.039,Z 860.977,A -85,B 0,C 180,E1 10223.66,E2 10223.66} C_VEL
LIN {X 0,Y 420.616,Z 830.827,A -85,B 0,C 180,E1 10227.326,E2 10227.326} C_VEL
LIN {X 0,Y 425.967,Z 797.074,A -85,B 0,C 180,E1 10230.225,E2 10230.225} C_VEL
LIN {X 0,Y 429.493,Z 763.931,A -85,B 0,C 180,E1 10232.253,E2 10232.253} C_VEL
LIN {X 0,Y 416.594,Z 731.651,A -85,B 0,C 180,E1 10235.336,E2 10235.336} C_VEL
LIN {X 0,Y 401.554,Z 703.444,A -85,B 0,C 180,E1 10238.221,E2 10238.221} C_VEL
LIN {X 0,Y 401.496,Z 702.53,A -85,B 0,C 180,E1 10238.487,E2 10238.487} C_VEL
LIN {X 0,Y 401.802,Z 702.53,A -85,B 0,C 180,E1 10244.78,E2 10244.78} C_VEL
LIN {X 0,Y 401.961,Z 702.53,A -85,B 0,C 180,E1 10251.383,E2 10251.383} C_VEL
LIN {X 0,Y 402.181,Z 702.53,A -85,B 0,C 180,E1 10257.867,E2 10257.867} C_VEL
LIN {X 0,Y 402.4,Z 702.53,A -85,B 0,C 180,E1 10262.166,E2 10262.166} C_VEL
LIN {X 0,Y 401.89,Z 702.53,A -85,B 0,C 180,E1 10268.653,E2 10268.653} C_VEL
LIN {X 0,Y 401.633,Z 702.53,A -85,B 0,C 180,E1 10275.263,E2 10275.263} C_VEL
LIN {X 0,Y 401.366,Z 702.53,A -85,B 0,C 180,E1 10282.098,E2 10282.098} C_VEL
